# B&R Automation Studio project Mapp6D_Demo
Automation Studio 4.10.3.60 SP; technology packages: mapp6D 1.1.0, mappView 5.12.1

## Configuration Config1

CPU X20CP1685, AutomationRuntime C4.90, Build 4.1.2, Safety 0.0, Vc V4.72.3

### Task classes (Cpu.sw)
```
Cyclic#4:
  Macro <- Macro.prg
  ShuttleGro <- ShuttleGroup.prg
  VirtualShu <- VirtualShuttle1.prg
  Planet <- Planet.prg
Binaries: FWRules, udbdef, TCData, arcoal, arflatprv, arsvcreg, arconfig, User, Role, sysconf, iomap, asfw, ashwac, ashwd, Config_2, Config_1
Libraries: McBase, brsystem, runtime, AsBrStr, McAcp6D, astime, asieccon, fileio
```

### Hardware
```
8YFLM01.0000.00I-1 : 8YFLM01.0000.00I-1 v0.0.0.1  [PLK1 -> X20CP1685.IF3 (NodeNumber=50) [Cable Type=PowerlinkCable, Length=10, Version=1.0.0.3]]
  Supervision = off
X20CP1685 : X20CP1685 v1.4.0.0
  Connector IF2:
    ActivateDevice = 1
    Mode = Manual
    InternetAddress = 192.168.10.7
    SubnetMask = 255.255.255.0
    ActivateSnmp = 2
  Connector IF3:
    CycleTime = 1000
  ConfigurationID = mapp6d_SampleProject_Config1
  UserPartitionSize = 10
  TimerDeviceType = EPLX2X
  TimerDevice = X20CP1685.IF3
  TaskClassIdleTime = 2000
  Cyclic1Duration = 1000
  Cyclic1Tolerance = 0
  Cyclic3Duration = 52000
  Cyclic3Tolerance = 52000
  Cyclic5Duration = 198000
  Cyclic5Tolerance = 198000
  Cyclic7Duration = 1002000
  Cyclic7Tolerance = 1002000
  FileDevice1
  FileDeviceName1 = 6DData
  FileDevicePath1 = C:\6DData
  FtpUser1
  FtpUsername1 = admin
  FtpUserPassword1 = dNmF8ZjP+LmBsEglWtmW9suMlO0FNzgHVeilX4YjqJw=
  FtpUserSalt1 = G7mT75Ku
  FTPAccessRight1 = 0
  FTPdevice1 = ALL
```

### Config_1.assembly6d - X20CP1685/mapp6D/Config_1.assembly6d
```
Element gAssembly6D_1 (Type=assembly6d)
  Simulation6D = SimOn
  Shuttles:
    MaxShuttleCount = 2
    ShuttleIDMode = RealTimeID
    DefaultPosition:
      DefZ = 1.0
      DefRx = 0
      DefRy = 0
      DefRz = 0
    Limits:
      InPlaneLimits:
        InPlaneVelLim = 2
        InPlaneAccLim = 20
        InPlaneEmergDec = 20
      ShortAxLim:
        ShortAxAccLim:
          AccZLim = 10.0
          AccRxLim = 10.0
          AccRyLim = 10.0
          AccRzLim = 10.0
        ShortAxVelLim:
          VelZLim = 0.15
          VelRxLim = 0.1
          VelRyLim = 0.1
          VelRzLim = 0.3
  CyclicChannel6D:
    ReadChannel:
      Xaxis = TRUE
      Yaxis = TRUE
      Zaxis = TRUE
      Rxaxis = TRUE
      Ryaxis = TRUE
      Rzaxis = TRUE
  Fieldbus6D:
    SyncMode6D = ExternalPlkSync
    NodeNumber = 50
  IOMapp:
    Input = ::gComm6D_IN
    Output = ::gComm6D_OUT
  Layout:
    Layout6D[1] = Layout6D_1
```

### Config_2.layout6d - X20CP1685/mapp6D/Config_2.layout6d
```
Element Layout6D_1 (Type=layout6d)
  Segments:
    SegRow = 2
    SegCol = 1
    Segment[1]:
      X = 0
      Y = 0
      Name
      IsMaster = True
    Segment[2]:
      X = 0
      Y = 1
      Name
      IsMaster = False
```

## Configuration Config2

CPU 5APC2100.BY44-000, AutomationRuntime D4.83, Build 4.1.2, Safety 0.0, Vc V4.72.3

### Task classes (Cpu.sw)
```
Cyclic#1 (cycle 1000 us, tolerance 0 us):
  MainCtrl <- MainCtrl.prg
Cyclic#2:
  Macro <- Macro.prg
Cyclic#8 (cycle 5000 us):
  HMI <- HMI.prg
Binaries: FWRules, udbdef, TCData, arcoal, arflatprv, arsvcreg, mvLoader, arconfig, User, Role, sysconf, iomap, asfw, ashwac, ashwd, Config_2, Config_1
Libraries: McBase, brsystem, runtime, AsBrStr, McAcp6D, brdkSTR, MTLookUp, sys_lib, standard, astime, asieccon, fileio, arssl
```

### Hardware
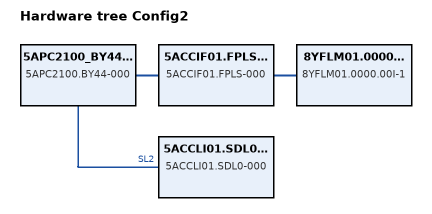
```
5ACCIF01.FPLS-000 : 5ACCIF01.FPLS-000 v2.6.1.0  [SL -> 5APC2100_BY44_000.SL1]
  Connector IF1:
    CycleTime = 1000
5ACCLI01.SDL0-000 : 5ACCLI01.SDL0-000 v2.0.0.0  [SL -> 5APC2100_BY44_000.SL2]
5APC2100_BY44_000 : 5APC2100.BY44-000 v2.1.0.0
  Connector IF3:
    AssignedOperatingSystem = ARemb
    ActivateDevice = 1
    Mode = Manual
    InternetAddress = 192.168.10.7
    SubnetMask = 255.255.255.0
    ActivateSnmp = 2
  Connector IF4:
    AssignedOperatingSystem = ARemb
    ActivateDevice = 1
    Mode = DHCP Server
    InternetAddress = 192.168.0.2
    SubnetMask = 255.255.255.0
    Lease1
    LeaseName1 = 6d_Demo
    LeaseStartAddress1 = 192.168.0.100
    LeaseStopAddress1 = 192.168.0.150
    LeaseSubnetMask1 = 255.255.255.0
  Connector IF5:
    AssignedOperatingSystem = ARemb
  Connector IF6:
    AssignedOperatingSystem = ARemb
  ConfigurationID = mapp6d_SampleProject_Config1
  UserPartitionSize = 10
  UserRamDevice = PCI.1.PPC21xx.SRAM
  UserRamSize = 5000
  RemMemDevice = PCI.1.PPC21xx.SRAM
  RemMemSize = 5000
  RemanentGlobalPvSize = 1000
  TimerDeviceType = EPLX2X
  TimerDevice = 5ACCIF01.FPLS-000.IF1
  TaskClassIdleTime = 2000
  Cyclic1Duration = 1000
  Cyclic1Tolerance = 0
  Cyclic3Duration = 52000
  Cyclic3Tolerance = 52000
  Cyclic5Duration = 198000
  Cyclic5Tolerance = 198000
  Cyclic7Duration = 1002000
  Cyclic7Tolerance = 1002000
  Cyclic8Duration = 5000
  FileDevice1
  FileDeviceName1 = 6DData
  FileDevicePath1 = F:
  FtpUser1
  FtpUsername1 = admin
  FtpUserPassword1 = dNmF8ZjP+LmBsEglWtmW9suMlO0FNzgHVeilX4YjqJw=
  FtpUserSalt1 = G7mT75Ku
  FTPAccessRight1 = 0
  FTPdevice1 = ALL
  ActivateOpcUa = 1
  OpcUaInformationModels_PV_Version = 1
8YFLM01.0000.00I-1 : 8YFLM01.0000.00I-1 v0.0.0.1  [PLK1 -> 5ACCIF01.FPLS-000.IF1 (NodeNumber=50) [Cable Type=PowerlinkCable, Length=10, Version=1.0.0.3]]
  Supervision = off
```

### IoMap.iom - 5APC2100_BY44_000/IoMap.iom
```iecst
VAR_CONFIG
	::gComm6D_IN.Array[0] AT %IW."8YFLM01.0000.00I-1".EPL_FB_IN_0_I2007_S01;
	::gComm6D_IN.Array[1] AT %IW."8YFLM01.0000.00I-1".EPL_FB_IN_1_I2007_S02;
	::gComm6D_IN.Array[2] AT %IW."8YFLM01.0000.00I-1".EPL_FB_IN_2_I2007_S03;
	::gComm6D_IN.Array[3] AT %IW."8YFLM01.0000.00I-1".EPL_FB_IN_3_I2007_S04;
	::gComm6D_IN.Array[4] AT %IW."8YFLM01.0000.00I-1".EPL_FB_IN_4_I2007_S05;
	::gComm6D_IN.Array[5] AT %IW."8YFLM01.0000.00I-1".EPL_FB_IN_5_I2007_S06;
	::gComm6D_IN.Array[6] AT %IW."8YFLM01.0000.00I-1".EPL_FB_IN_6_I2007_S07;
	::gComm6D_IN.Array[7] AT %IW."8YFLM01.0000.00I-1".EPL_FB_IN_7_I2007_S08;
	::gComm6D_IN.Array[8] AT %IW."8YFLM01.0000.00I-1".EPL_FB_IN_8_I2007_S09;
	::gComm6D_IN.Array[9] AT %IW."8YFLM01.0000.00I-1".EPL_FB_IN_9_I2007_S0A;
	::gComm6D_IN.Array[10] AT %IW."8YFLM01.0000.00I-1".EPL_FB_IN_10_I2007_S0B;
	::gComm6D_IN.Array[11] AT %IW."8YFLM01.0000.00I-1".EPL_FB_IN_11_I2007_S0C;
	::gComm6D_IN.Array[12] AT %IW."8YFLM01.0000.00I-1".EPL_FB_IN_12_I2007_S0D;
	::gComm6D_IN.Array[13] AT %IW."8YFLM01.0000.00I-1".EPL_FB_IN_13_I2007_S0E;
	::gComm6D_IN.Array[14] AT %IW."8YFLM01.0000.00I-1".EPL_FB_IN_14_I2007_S0F;
	::gComm6D_IN.Array[15] AT %IW."8YFLM01.0000.00I-1".EPL_FB_IN_15_I2007_S10;
	::gComm6D_IN.Array[16] AT %IW."8YFLM01.0000.00I-1".EPL_FB_IN_16_I2007_S11;
	::gComm6D_IN.Array[17] AT %IW."8YFLM01.0000.00I-1".EPL_FB_IN_17_I2007_S12;
	::gComm6D_IN.Array[18] AT %IW."8YFLM01.0000.00I-1".EPL_FB_IN_18_I2007_S13;
	::gComm6D_IN.Array[19] AT %IW."8YFLM01.0000.00I-1".EPL_FB_IN_19_I2007_S14;
	::gComm6D_IN.Array[20] AT %IW."8YFLM01.0000.00I-1".EPL_FB_IN_20_I2007_S15;
	::gComm6D_IN.Array[21] AT %IW."8YFLM01.0000.00I-1".EPL_FB_IN_21_I2007_S16;
	::gComm6D_IN.Array[22] AT %IW."8YFLM01.0000.00I-1".EPL_FB_IN_22_I2007_S17;
	::gComm6D_IN.Array[23] AT %IW."8YFLM01.0000.00I-1".EPL_FB_IN_23_I2007_S18;
	::gComm6D_IN.Array[24] AT %IW."8YFLM01.0000.00I-1".EPL_FB_IN_24_I2007_S19;
	::gComm6D_IN.Array[25] AT %IW."8YFLM01.0000.00I-1".EPL_FB_IN_25_I2007_S1A;
	::gComm6D_IN.Array[26] AT %IW."8YFLM01.0000.00I-1".EPL_FB_IN_26_I2007_S1B;
	::gComm6D_IN.Array[27] AT %IW."8YFLM01.0000.00I-1".EPL_FB_IN_27_I2007_S1C;
	::gComm6D_IN.Array[28] AT %IW."8YFLM01.0000.00I-1".EPL_FB_IN_28_I2007_S1D;
	::gComm6D_IN.Array[29] AT %IW."8YFLM01.0000.00I-1".EPL_FB_IN_29_I2007_S1E;
	::gComm6D_IN.Array[30] AT %IW."8YFLM01.0000.00I-1".EPL_FB_IN_30_I2007_S1F;
	::gComm6D_IN.Array[31] AT %IW."8YFLM01.0000.00I-1".EPL_FB_IN_31_I2007_S20;
	::gComm6D_IN.Array[32] AT %IW."8YFLM01.0000.00I-1".EPL_FB_IN_32_I2007_S21;
	::gComm6D_IN.Array[33] AT %IW."8YFLM01.0000.00I-1".EPL_FB_IN_33_I2007_S22;
	::gComm6D_IN.Array[34] AT %IW."8YFLM01.0000.00I-1".EPL_FB_IN_34_I2007_S23;
	::gComm6D_IN.Array[35] AT %IW."8YFLM01.0000.00I-1".EPL_FB_IN_35_I2007_S24;
	::gComm6D_IN.Array[36] AT %IW."8YFLM01.0000.00I-1".EPL_FB_IN_36_I2007_S25;
	::gComm6D_IN.Array[37] AT %IW."8YFLM01.0000.00I-1".EPL_FB_IN_37_I2007_S26;
	::gComm6D_IN.Array[38] AT %IW."8YFLM01.0000.00I-1".EPL_FB_IN_38_I2007_S27;
	::gComm6D_IN.Array[39] AT %IW."8YFLM01.0000.00I-1".EPL_FB_IN_39_I2007_S28;
	::gComm6D_IN.Array[40] AT %IW."8YFLM01.0000.00I-1".EPL_FB_IN_40_I2007_S29;
	::gComm6D_IN.Array[41] AT %IW."8YFLM01.0000.00I-1".EPL_FB_IN_41_I2007_S2A;
	::gComm6D_IN.Array[42] AT %IW."8YFLM01.0000.00I-1".EPL_FB_IN_42_I2007_S2B;
	::gComm6D_IN.Array[43] AT %IW."8YFLM01.0000.00I-1".EPL_FB_IN_43_I2007_S2C;
	::gComm6D_IN.Array[44] AT %IW."8YFLM01.0000.00I-1".EPL_FB_IN_44_I2007_S2D;
	::gComm6D_IN.Array[45] AT %IW."8YFLM01.0000.00I-1".EPL_FB_IN_45_I2007_S2E;
	::gComm6D_IN.Array[46] AT %IW."8YFLM01.0000.00I-1".EPL_FB_IN_46_I2007_S2F;
	::gComm6D_IN.Array[47] AT %IW."8YFLM01.0000.00I-1".EPL_FB_IN_47_I2007_S30;
	::gComm6D_IN.Array[48] AT %IW."8YFLM01.0000.00I-1".EPL_FB_IN_48_I2007_S31;
	::gComm6D_IN.Array[49] AT %IW."8YFLM01.0000.00I-1".EPL_FB_IN_49_I2007_S32;
	::gComm6D_IN.Array[50] AT %IW."8YFLM01.0000.00I-1".EPL_FB_IN_50_I2007_S33;
	::gComm6D_IN.Array[51] AT %IW."8YFLM01.0000.00I-1".EPL_FB_IN_51_I2007_S34;
	::gComm6D_IN.Array[52] AT %IW."8YFLM01.0000.00I-1".EPL_FB_IN_52_I2007_S35;
	::gComm6D_IN.Array[53] AT %IW."8YFLM01.0000.00I-1".EPL_FB_IN_53_I2007_S36;
	::gComm6D_IN.Array[54] AT %IW."8YFLM01.0000.00I-1".EPL_FB_IN_54_I2007_S37;
	::gComm6D_IN.Array[55] AT %IW."8YFLM01.0000.00I-1".EPL_FB_IN_55_I2007_S38;
	::gComm6D_IN.Array[56] AT %IW."8YFLM01.0000.00I-1".EPL_FB_IN_56_I2007_S39;
	::gComm6D_IN.Array[57] AT %IW."8YFLM01.0000.00I-1".EPL_FB_IN_57_I2007_S3A;
	::gComm6D_IN.Array[58] AT %IW."8YFLM01.0000.00I-1".EPL_FB_IN_58_I2007_S3B;
	::gComm6D_IN.Array[59] AT %IW."8YFLM01.0000.00I-1".EPL_FB_IN_59_I2007_S3C;
	::gComm6D_IN.Array[60] AT %IW."8YFLM01.0000.00I-1".EPL_FB_IN_60_I2007_S3D;
	::gComm6D_IN.Array[61] AT %IW."8YFLM01.0000.00I-1".EPL_FB_IN_61_I2007_S3E;
	::gComm6D_IN.Array[62] AT %IW."8YFLM01.0000.00I-1".EPL_FB_IN_62_I2007_S3F;
	::gComm6D_IN.Array[63] AT %IW."8YFLM01.0000.00I-1".EPL_FB_IN_63_I2007_S40;
	::gComm6D_IN.Array[64] AT %IW."8YFLM01.0000.00I-1".EPL_FB_IN_64_I2007_S41;
	::gComm6D_IN.Array[65] AT %IW."8YFLM01.0000.00I-1".EPL_FB_IN_65_I2007_S42;
	::gComm6D_IN.Array[66] AT %IW."8YFLM01.0000.00I-1".EPL_FB_IN_66_I2007_S43;
	::gComm6D_IN.Array[67] AT %IW."8YFLM01.0000.00I-1".EPL_FB_IN_67_I2007_S44;
	::gComm6D_IN.Array[68] AT %IW."8YFLM01.0000.00I-1".EPL_FB_IN_68_I2007_S45;
	::gComm6D_IN.Array[69] AT %IW."8YFLM01.0000.00I-1".EPL_FB_IN_69_I2007_S46;
	::gComm6D_IN.Array[70] AT %IW."8YFLM01.0000.00I-1".EPL_FB_IN_70_I2007_S47;
	::gComm6D_IN.Array[71] AT %IW."8YFLM01.0000.00I-1".EPL_FB_IN_71_I2007_S48;
	::gComm6D_IN.Array[72] AT %IW."8YFLM01.0000.00I-1".EPL_FB_IN_72_I2007_S49;
	::gComm6D_IN.Array[73] AT %IW."8YFLM01.0000.00I-1".EPL_FB_IN_73_I2007_S4A;
	::gComm6D_IN.Array[74] AT %IW."8YFLM01.0000.00I-1".EPL_FB_IN_74_I2007_S4B;
	::gComm6D_IN.Array[75] AT %IW."8YFLM01.0000.00I-1".EPL_FB_IN_75_I2007_S4C;
	::gComm6D_IN.Array[76] AT %IW."8YFLM01.0000.00I-1".EPL_FB_IN_76_I2007_S4D;
	::gComm6D_IN.Array[77] AT %IW."8YFLM01.0000.00I-1".EPL_FB_IN_77_I2007_S4E;
	::gComm6D_IN.Array[78] AT %IW."8YFLM01.0000.00I-1".EPL_FB_IN_78_I2007_S4F;
	::gComm6D_IN.Array[79] AT %IW."8YFLM01.0000.00I-1".EPL_FB_IN_79_I2007_S50;
	::gComm6D_IN.Array[80] AT %IW."8YFLM01.0000.00I-1".EPL_FB_IN_80_I2007_S51;
	::gComm6D_IN.Array[81] AT %IW."8YFLM01.0000.00I-1".EPL_FB_IN_81_I2007_S52;
	::gComm6D_IN.Array[82] AT %IW."8YFLM01.0000.00I-1".EPL_FB_IN_82_I2007_S53;
	::gComm6D_IN.Array[83] AT %IW."8YFLM01.0000.00I-1".EPL_FB_IN_83_I2007_S54;
	::gComm6D_IN.Array[84] AT %IW."8YFLM01.0000.00I-1".EPL_FB_IN_84_I2007_S55;
	::gComm6D_IN.Array[85] AT %IW."8YFLM01.0000.00I-1".EPL_FB_IN_85_I2007_S56;
	::gComm6D_IN.Array[86] AT %IW."8YFLM01.0000.00I-1".EPL_FB_IN_86_I2007_S57;
	::gComm6D_IN.Array[87] AT %IW."8YFLM01.0000.00I-1".EPL_FB_IN_87_I2007_S58;
	::gComm6D_IN.Array[88] AT %IW."8YFLM01.0000.00I-1".EPL_FB_IN_88_I2007_S59;
	::gComm6D_IN.Array[89] AT %IW."8YFLM01.0000.00I-1".EPL_FB_IN_89_I2007_S5A;
	::gComm6D_IN.Array[90] AT %IW."8YFLM01.0000.00I-1".EPL_FB_IN_90_I2007_S5B;
	::gComm6D_IN.Array[91] AT %IW."8YFLM01.0000.00I-1".EPL_FB_IN_91_I2007_S5C;
	::gComm6D_IN.Array[92] AT %IW."8YFLM01.0000.00I-1".EPL_FB_IN_92_I2007_S5D;
	::gComm6D_IN.Array[93] AT %IW."8YFLM01.0000.00I-1".EPL_FB_IN_93_I2007_S5E;
	::gComm6D_IN.Array[94] AT %IW."8YFLM01.0000.00I-1".EPL_FB_IN_94_I2007_S5F;
	::gComm6D_IN.Array[95] AT %IW."8YFLM01.0000.00I-1".EPL_FB_IN_95_I2007_S60;
	::gComm6D_IN.Array[96] AT %IW."8YFLM01.0000.00I-1".EPL_FB_IN_96_I2007_S61;
	::gComm6D_IN.Array[97] AT %IW."8YFLM01.0000.00I-1".EPL_FB_IN_97_I2007_S62;
	::gComm6D_IN.Array[98] AT %IW."8YFLM01.0000.00I-1".EPL_FB_IN_98_I2007_S63;
	::gComm6D_IN.Array[99] AT %IW."8YFLM01.0000.00I-1".EPL_FB_IN_99_I2007_S64;
	::gComm6D_IN.Array[100] AT %IW."8YFLM01.0000.00I-1".EPL_FB_IN_100_I2007_S65;
	::gComm6D_IN.Array[101] AT %IW."8YFLM01.0000.00I-1".EPL_FB_IN_101_I2007_S66;
	::gComm6D_IN.Array[102] AT %IW."8YFLM01.0000.00I-1".EPL_FB_IN_102_I2007_S67;
	::gComm6D_IN.Array[103] AT %IW."8YFLM01.0000.00I-1".EPL_FB_IN_103_I2007_S68;
	::gComm6D_IN.Array[104] AT %IW."8YFLM01.0000.00I-1".EPL_FB_IN_104_I2007_S69;
	::gComm6D_IN.Array[105] AT %IW."8YFLM01.0000.00I-1".EPL_FB_IN_105_I2007_S6A;
	::gComm6D_IN.Array[106] AT %IW."8YFLM01.0000.00I-1".EPL_FB_IN_106_I2007_S6B;
	::gComm6D_IN.Array[107] AT %IW."8YFLM01.0000.00I-1".EPL_FB_IN_107_I2007_S6C;
	::gComm6D_IN.Array[108] AT %IW."8YFLM01.0000.00I-1".EPL_FB_IN_108_I2007_S6D;
	::gComm6D_IN.Array[109] AT %IW."8YFLM01.0000.00I-1".EPL_FB_IN_109_I2007_S6E;
	::gComm6D_IN.Array[110] AT %IW."8YFLM01.0000.00I-1".EPL_FB_IN_110_I2007_S6F;
	::gComm6D_IN.Array[111] AT %IW."8YFLM01.0000.00I-1".EPL_FB_IN_111_I2007_S70;
	::gComm6D_IN.Array[112] AT %IW."8YFLM01.0000.00I-1".EPL_FB_IN_112_I2007_S71;
	::gComm6D_IN.Array[113] AT %IW."8YFLM01.0000.00I-1".EPL_FB_IN_113_I2007_S72;
	::gComm6D_IN.Array[114] AT %IW."8YFLM01.0000.00I-1".EPL_FB_IN_114_I2007_S73;
	::gComm6D_IN.Array[115] AT %IW."8YFLM01.0000.00I-1".EPL_FB_IN_115_I2007_S74;
	::gComm6D_IN.Array[116] AT %IW."8YFLM01.0000.00I-1".EPL_FB_IN_116_I2007_S75;
	::gComm6D_IN.Array[117] AT %IW."8YFLM01.0000.00I-1".EPL_FB_IN_117_I2007_S76;
	::gComm6D_IN.Array[118] AT %IW."8YFLM01.0000.00I-1".EPL_FB_IN_118_I2007_S77;
	::gComm6D_IN.Array[119] AT %IW."8YFLM01.0000.00I-1".EPL_FB_IN_119_I2007_S78;
	::gComm6D_IN.Array[120] AT %IW."8YFLM01.0000.00I-1".EPL_FB_IN_120_I2007_S79;
	::gComm6D_IN.Array[121] AT %IW."8YFLM01.0000.00I-1".EPL_FB_IN_121_I2007_S7A;
	::gComm6D_IN.Array[122] AT %IW."8YFLM01.0000.00I-1".EPL_FB_IN_122_I2007_S7B;
	::gComm6D_IN.Array[123] AT %IW."8YFLM01.0000.00I-1".EPL_FB_IN_123_I2007_S7C;
	::gComm6D_IN.Array[124] AT %IW."8YFLM01.0000.00I-1".EPL_FB_IN_124_I2007_S7D;
	::gComm6D_IN.Array[125] AT %IW."8YFLM01.0000.00I-1".EPL_FB_IN_125_I2007_S7E;
	::gComm6D_IN.Array[126] AT %IW."8YFLM01.0000.00I-1".EPL_FB_IN_126_I2007_S7F;
	::gComm6D_IN.Array[127] AT %IW."8YFLM01.0000.00I-1".EPL_FB_IN_127_I2007_S80;
	::gComm6D_IN.Array[128] AT %IW."8YFLM01.0000.00I-1".EPL_FB_IN_128_I2007_S81;
	::gComm6D_IN.Array[129] AT %IW."8YFLM01.0000.00I-1".EPL_FB_IN_129_I2007_S82;
	::gComm6D_IN.Array[130] AT %IW."8YFLM01.0000.00I-1".EPL_FB_IN_130_I2007_S83;
	::gComm6D_IN.Array[131] AT %IW."8YFLM01.0000.00I-1".EPL_FB_IN_131_I2007_S84;
	::gComm6D_IN.Array[132] AT %IW."8YFLM01.0000.00I-1".EPL_FB_IN_132_I2007_S85;
	::gComm6D_IN.Array[133] AT %IW."8YFLM01.0000.00I-1".EPL_FB_IN_133_I2007_S86;
	::gComm6D_IN.Array[134] AT %IW."8YFLM01.0000.00I-1".EPL_FB_IN_134_I2007_S87;
	::gComm6D_IN.Array[135] AT %IW."8YFLM01.0000.00I-1".EPL_FB_IN_135_I2007_S88;
	::gComm6D_IN.Array[136] AT %IW."8YFLM01.0000.00I-1".EPL_FB_IN_136_I2007_S89;
	::gComm6D_IN.Array[137] AT %IW."8YFLM01.0000.00I-1".EPL_FB_IN_137_I2007_S8A;
	::gComm6D_IN.Array[138] AT %IW."8YFLM01.0000.00I-1".EPL_FB_IN_138_I2007_S8B;
	::gComm6D_IN.Array[139] AT %IW."8YFLM01.0000.00I-1".EPL_FB_IN_139_I2007_S8C;
	::gComm6D_IN.Array[140] AT %IW."8YFLM01.0000.00I-1".EPL_FB_IN_140_I2007_S8D;
	::gComm6D_IN.Array[141] AT %IW."8YFLM01.0000.00I-1".EPL_FB_IN_141_I2007_S8E;
	::gComm6D_IN.Array[142] AT %IW."8YFLM01.0000.00I-1".EPL_FB_IN_142_I2007_S8F;
	::gComm6D_IN.Array[143] AT %IW."8YFLM01.0000.00I-1".EPL_FB_IN_143_I2007_S90;
	::gComm6D_IN.Array[144] AT %IW."8YFLM01.0000.00I-1".EPL_FB_IN_144_I2007_S91;
	::gComm6D_IN.Array[145] AT %IW."8YFLM01.0000.00I-1".EPL_FB_IN_145_I2007_S92;
	::gComm6D_IN.Array[146] AT %IW."8YFLM01.0000.00I-1".EPL_FB_IN_146_I2007_S93;
	::gComm6D_IN.Array[147] AT %IW."8YFLM01.0000.00I-1".EPL_FB_IN_147_I2007_S94;
	::gComm6D_IN.Array[148] AT %IW."8YFLM01.0000.00I-1".EPL_FB_IN_148_I2007_S95;
	::gComm6D_IN.Array[149] AT %IW."8YFLM01.0000.00I-1".EPL_FB_IN_149_I2007_S96;
	::gComm6D_IN.Array[150] AT %IW."8YFLM01.0000.00I-1".EPL_FB_IN_150_I2007_S97;
	::gComm6D_IN.Array[151] AT %IW."8YFLM01.0000.00I-1".EPL_FB_IN_151_I2007_S98;
	::gComm6D_IN.Array[152] AT %IW."8YFLM01.0000.00I-1".EPL_FB_IN_152_I2007_S99;
	::gComm6D_IN.Array[153] AT %IW."8YFLM01.0000.00I-1".EPL_FB_IN_153_I2007_S9A;
	::gComm6D_IN.Array[154] AT %IW."8YFLM01.0000.00I-1".EPL_FB_IN_154_I2007_S9B;
	::gComm6D_IN.Array[155] AT %IW."8YFLM01.0000.00I-1".EPL_FB_IN_155_I2007_S9C;
	::gComm6D_IN.Array[156] AT %IW."8YFLM01.0000.00I-1".EPL_FB_IN_156_I2007_S9D;
	::gComm6D_IN.Array[157] AT %IW."8YFLM01.0000.00I-1".EPL_FB_IN_157_I2007_S9E;
	::gComm6D_IN.Array[158] AT %IW."8YFLM01.0000.00I-1".EPL_FB_IN_158_I2007_S9F;
	::gComm6D_IN.Array[159] AT %IW."8YFLM01.0000.00I-1".EPL_FB_IN_159_I2007_SA0;
	::gComm6D_IN.Array[160] AT %IW."8YFLM01.0000.00I-1".EPL_FB_IN_160_I2007_SA1;
	::gComm6D_IN.Array[161] AT %IW."8YFLM01.0000.00I-1".EPL_FB_IN_161_I2007_SA2;
	::gComm6D_IN.Array[162] AT %IW."8YFLM01.0000.00I-1".EPL_FB_IN_162_I2007_SA3;
	::gComm6D_IN.Array[163] AT %IW."8YFLM01.0000.00I-1".EPL_FB_IN_163_I2007_SA4;
	::gComm6D_IN.Array[164] AT %IW."8YFLM01.0000.00I-1".EPL_FB_IN_164_I2007_SA5;
	::gComm6D_IN.Array[165] AT %IW."8YFLM01.0000.00I-1".EPL_FB_IN_165_I2007_SA6;
	::gComm6D_IN.Array[166] AT %IW."8YFLM01.0000.00I-1".EPL_FB_IN_166_I2007_SA7;
	::gComm6D_IN.Array[167] AT %IW."8YFLM01.0000.00I-1".EPL_FB_IN_167_I2007_SA8;
	::gComm6D_IN.Array[168] AT %IW."8YFLM01.0000.00I-1".EPL_FB_IN_168_I2007_SA9;
	::gComm6D_IN.Array[169] AT %IW."8YFLM01.0000.00I-1".EPL_FB_IN_169_I2007_SAA;
	::gComm6D_IN.Array[170] AT %IW."8YFLM01.0000.00I-1".EPL_FB_IN_170_I2007_SAB;
	::gComm6D_IN.Array[171] AT %IW."8YFLM01.0000.00I-1".EPL_FB_IN_171_I2007_SAC;
	::gComm6D_IN.Array[172] AT %IW."8YFLM01.0000.00I-1".EPL_FB_IN_172_I2007_SAD;
	::gComm6D_IN.Array[173] AT %IW."8YFLM01.0000.00I-1".EPL_FB_IN_173_I2007_SAE;
	::gComm6D_IN.Array[174] AT %IW."8YFLM01.0000.00I-1".EPL_FB_IN_174_I2007_SAF;
	::gComm6D_IN.Array[175] AT %IW."8YFLM01.0000.00I-1".EPL_FB_IN_175_I2007_SB0;
	::gComm6D_IN.Array[176] AT %IW."8YFLM01.0000.00I-1".EPL_FB_IN_176_I2007_SB1;
	::gComm6D_IN.Array[177] AT %IW."8YFLM01.0000.00I-1".EPL_FB_IN_177_I2007_SB2;
	::gComm6D_IN.Array[178] AT %IW."8YFLM01.0000.00I-1".EPL_FB_IN_178_I2007_SB3;
	::gComm6D_IN.Array[179] AT %IW."8YFLM01.0000.00I-1".EPL_FB_IN_179_I2007_SB4;
	::gComm6D_IN.Array[180] AT %IW."8YFLM01.0000.00I-1".EPL_FB_IN_180_I2007_SB5;
	::gComm6D_IN.Array[181] AT %IW."8YFLM01.0000.00I-1".EPL_FB_IN_181_I2007_SB6;
	::gComm6D_IN.Array[182] AT %IW."8YFLM01.0000.00I-1".EPL_FB_IN_182_I2007_SB7;
	::gComm6D_IN.Array[183] AT %IW."8YFLM01.0000.00I-1".EPL_FB_IN_183_I2007_SB8;
	::gComm6D_IN.Array[184] AT %IW."8YFLM01.0000.00I-1".EPL_FB_IN_184_I2007_SB9;
	::gComm6D_IN.Array[185] AT %IW."8YFLM01.0000.00I-1".EPL_FB_IN_185_I2007_SBA;
	::gComm6D_IN.Array[186] AT %IW."8YFLM01.0000.00I-1".EPL_FB_IN_186_I2007_SBB;
	::gComm6D_IN.Array[187] AT %IW."8YFLM01.0000.00I-1".EPL_FB_IN_187_I2007_SBC;
	::gComm6D_IN.Array[188] AT %IW."8YFLM01.0000.00I-1".EPL_FB_IN_188_I2007_SBD;
	::gComm6D_IN.Array[189] AT %IW."8YFLM01.0000.00I-1".EPL_FB_IN_189_I2007_SBE;
	::gComm6D_IN.Array[190] AT %IW."8YFLM01.0000.00I-1".EPL_FB_IN_190_I2007_SBF;
	::gComm6D_IN.Array[191] AT %IW."8YFLM01.0000.00I-1".EPL_FB_IN_191_I2007_SC0;
	::gComm6D_IN.Array[192] AT %IW."8YFLM01.0000.00I-1".EPL_FB_IN_192_I2007_SC1;
	::gComm6D_IN.Array[193] AT %IW."8YFLM01.0000.00I-1".EPL_FB_IN_193_I2007_SC2;
	::gComm6D_IN.Array[194] AT %IW."8YFLM01.0000.00I-1".EPL_FB_IN_194_I2007_SC3;
	::gComm6D_IN.Array[195] AT %IW."8YFLM01.0000.00I-1".EPL_FB_IN_195_I2007_SC4;
	::gComm6D_IN.Array[196] AT %IW."8YFLM01.0000.00I-1".EPL_FB_IN_196_I2007_SC5;
	::gComm6D_IN.Array[197] AT %IW."8YFLM01.0000.00I-1".EPL_FB_IN_197_I2007_SC6;
	::gComm6D_IN.Array[198] AT %IW."8YFLM01.0000.00I-1".EPL_FB_IN_198_I2007_SC7;
	::gComm6D_IN.Array[199] AT %IW."8YFLM01.0000.00I-1".EPL_FB_IN_199_I2007_SC8;
	::gComm6D_OUT.Array[0] AT %QW."8YFLM01.0000.00I-1".EPL_FB_OUT_0_I2008_S01Out;
	::gComm6D_OUT.Array[1] AT %QW."8YFLM01.0000.00I-1".EPL_FB_OUT_1_I2008_S02Out;
	::gComm6D_OUT.Array[2] AT %QW."8YFLM01.0000.00I-1".EPL_FB_OUT_2_I2008_S03Out;
	::gComm6D_OUT.Array[3] AT %QW."8YFLM01.0000.00I-1".EPL_FB_OUT_3_I2008_S04Out;
	::gComm6D_OUT.Array[4] AT %QW."8YFLM01.0000.00I-1".EPL_FB_OUT_4_I2008_S05Out;
	::gComm6D_OUT.Array[5] AT %QW."8YFLM01.0000.00I-1".EPL_FB_OUT_5_I2008_S06Out;
	::gComm6D_OUT.Array[6] AT %QW."8YFLM01.0000.00I-1".EPL_FB_OUT_6_I2008_S07Out;
	::gComm6D_OUT.Array[7] AT %QW."8YFLM01.0000.00I-1".EPL_FB_OUT_7_I2008_S08Out;
	::gComm6D_OUT.Array[8] AT %QW."8YFLM01.0000.00I-1".EPL_FB_OUT_8_I2008_S09Out;
	::gComm6D_OUT.Array[9] AT %QW."8YFLM01.0000.00I-1".EPL_FB_OUT_9_I2008_S0AOut;
	::gComm6D_OUT.Array[10] AT %QW."8YFLM01.0000.00I-1".EPL_FB_OUT_10_I2008_S0BOut;
	::gComm6D_OUT.Array[11] AT %QW."8YFLM01.0000.00I-1".EPL_FB_OUT_11_I2008_S0COut;
	::gComm6D_OUT.Array[12] AT %QW."8YFLM01.0000.00I-1".EPL_FB_OUT_12_I2008_S0DOut;
	::gComm6D_OUT.Array[13] AT %QW."8YFLM01.0000.00I-1".EPL_FB_OUT_13_I2008_S0EOut;
	::gComm6D_OUT.Array[14] AT %QW."8YFLM01.0000.00I-1".EPL_FB_OUT_14_I2008_S0FOut;
	::gComm6D_OUT.Array[15] AT %QW."8YFLM01.0000.00I-1".EPL_FB_OUT_15_I2008_S10Out;
	::gComm6D_OUT.Array[16] AT %QW."8YFLM01.0000.00I-1".EPL_FB_OUT_16_I2008_S11Out;
	::gComm6D_OUT.Array[17] AT %QW."8YFLM01.0000.00I-1".EPL_FB_OUT_17_I2008_S12Out;
	::gComm6D_OUT.Array[18] AT %QW."8YFLM01.0000.00I-1".EPL_FB_OUT_18_I2008_S13Out;
	::gComm6D_OUT.Array[19] AT %QW."8YFLM01.0000.00I-1".EPL_FB_OUT_19_I2008_S14Out;
	::gComm6D_OUT.Array[20] AT %QW."8YFLM01.0000.00I-1".EPL_FB_OUT_20_I2008_S15Out;
	::gComm6D_OUT.Array[21] AT %QW."8YFLM01.0000.00I-1".EPL_FB_OUT_21_I2008_S16Out;
	::gComm6D_OUT.Array[22] AT %QW."8YFLM01.0000.00I-1".EPL_FB_OUT_22_I2008_S17Out;
	::gComm6D_OUT.Array[23] AT %QW."8YFLM01.0000.00I-1".EPL_FB_OUT_23_I2008_S18Out;
	::gComm6D_OUT.Array[24] AT %QW."8YFLM01.0000.00I-1".EPL_FB_OUT_24_I2008_S19Out;
	::gComm6D_OUT.Array[25] AT %QW."8YFLM01.0000.00I-1".EPL_FB_OUT_25_I2008_S1AOut;
	::gComm6D_OUT.Array[26] AT %QW."8YFLM01.0000.00I-1".EPL_FB_OUT_26_I2008_S1BOut;
	::gComm6D_OUT.Array[27] AT %QW."8YFLM01.0000.00I-1".EPL_FB_OUT_27_I2008_S1COut;
	::gComm6D_OUT.Array[28] AT %QW."8YFLM01.0000.00I-1".EPL_FB_OUT_28_I2008_S1DOut;
	::gComm6D_OUT.Array[29] AT %QW."8YFLM01.0000.00I-1".EPL_FB_OUT_29_I2008_S1EOut;
	::gComm6D_OUT.Array[30] AT %QW."8YFLM01.0000.00I-1".EPL_FB_OUT_30_I2008_S1FOut;
	::gComm6D_OUT.Array[31] AT %QW."8YFLM01.0000.00I-1".EPL_FB_OUT_31_I2008_S20Out;
	::gComm6D_OUT.Array[32] AT %QW."8YFLM01.0000.00I-1".EPL_FB_OUT_32_I2008_S21Out;
	::gComm6D_OUT.Array[33] AT %QW."8YFLM01.0000.00I-1".EPL_FB_OUT_33_I2008_S22Out;
	::gComm6D_OUT.Array[34] AT %QW."8YFLM01.0000.00I-1".EPL_FB_OUT_34_I2008_S23Out;
	::gComm6D_OUT.Array[35] AT %QW."8YFLM01.0000.00I-1".EPL_FB_OUT_35_I2008_S24Out;
	::gComm6D_OUT.Array[36] AT %QW."8YFLM01.0000.00I-1".EPL_FB_OUT_36_I2008_S25Out;
	::gComm6D_OUT.Array[37] AT %QW."8YFLM01.0000.00I-1".EPL_FB_OUT_37_I2008_S26Out;
	::gComm6D_OUT.Array[38] AT %QW."8YFLM01.0000.00I-1".EPL_FB_OUT_38_I2008_S27Out;
	::gComm6D_OUT.Array[39] AT %QW."8YFLM01.0000.00I-1".EPL_FB_OUT_39_I2008_S28Out;
	::gComm6D_OUT.Array[40] AT %QW."8YFLM01.0000.00I-1".EPL_FB_OUT_40_I2008_S29Out;
	::gComm6D_OUT.Array[41] AT %QW."8YFLM01.0000.00I-1".EPL_FB_OUT_41_I2008_S2AOut;
	::gComm6D_OUT.Array[42] AT %QW."8YFLM01.0000.00I-1".EPL_FB_OUT_42_I2008_S2BOut;
	::gComm6D_OUT.Array[43] AT %QW."8YFLM01.0000.00I-1".EPL_FB_OUT_43_I2008_S2COut;
	::gComm6D_OUT.Array[44] AT %QW."8YFLM01.0000.00I-1".EPL_FB_OUT_44_I2008_S2DOut;
	::gComm6D_OUT.Array[45] AT %QW."8YFLM01.0000.00I-1".EPL_FB_OUT_45_I2008_S2EOut;
	::gComm6D_OUT.Array[46] AT %QW."8YFLM01.0000.00I-1".EPL_FB_OUT_46_I2008_S2FOut;
	::gComm6D_OUT.Array[47] AT %QW."8YFLM01.0000.00I-1".EPL_FB_OUT_47_I2008_S30Out;
	::gComm6D_OUT.Array[48] AT %QW."8YFLM01.0000.00I-1".EPL_FB_OUT_48_I2008_S31Out;
	::gComm6D_OUT.Array[49] AT %QW."8YFLM01.0000.00I-1".EPL_FB_OUT_49_I2008_S32Out;
	::gComm6D_OUT.Array[50] AT %QW."8YFLM01.0000.00I-1".EPL_FB_OUT_50_I2008_S33Out;
	::gComm6D_OUT.Array[51] AT %QW."8YFLM01.0000.00I-1".EPL_FB_OUT_51_I2008_S34Out;
	::gComm6D_OUT.Array[52] AT %QW."8YFLM01.0000.00I-1".EPL_FB_OUT_52_I2008_S35Out;
	::gComm6D_OUT.Array[53] AT %QW."8YFLM01.0000.00I-1".EPL_FB_OUT_53_I2008_S36Out;
	::gComm6D_OUT.Array[54] AT %QW."8YFLM01.0000.00I-1".EPL_FB_OUT_54_I2008_S37Out;
	::gComm6D_OUT.Array[55] AT %QW."8YFLM01.0000.00I-1".EPL_FB_OUT_55_I2008_S38Out;
	::gComm6D_OUT.Array[56] AT %QW."8YFLM01.0000.00I-1".EPL_FB_OUT_56_I2008_S39Out;
	::gComm6D_OUT.Array[57] AT %QW."8YFLM01.0000.00I-1".EPL_FB_OUT_57_I2008_S3AOut;
	::gComm6D_OUT.Array[58] AT %QW."8YFLM01.0000.00I-1".EPL_FB_OUT_58_I2008_S3BOut;
	::gComm6D_OUT.Array[59] AT %QW."8YFLM01.0000.00I-1".EPL_FB_OUT_59_I2008_S3COut;
	::gComm6D_OUT.Array[60] AT %QW."8YFLM01.0000.00I-1".EPL_FB_OUT_60_I2008_S3DOut;
	::gComm6D_OUT.Array[61] AT %QW."8YFLM01.0000.00I-1".EPL_FB_OUT_61_I2008_S3EOut;
	::gComm6D_OUT.Array[62] AT %QW."8YFLM01.0000.00I-1".EPL_FB_OUT_62_I2008_S3FOut;
	::gComm6D_OUT.Array[63] AT %QW."8YFLM01.0000.00I-1".EPL_FB_OUT_63_I2008_S40Out;
	::gComm6D_OUT.Array[64] AT %QW."8YFLM01.0000.00I-1".EPL_FB_OUT_64_I2008_S41Out;
	::gComm6D_OUT.Array[65] AT %QW."8YFLM01.0000.00I-1".EPL_FB_OUT_65_I2008_S42Out;
	::gComm6D_OUT.Array[66] AT %QW."8YFLM01.0000.00I-1".EPL_FB_OUT_66_I2008_S43Out;
	::gComm6D_OUT.Array[67] AT %QW."8YFLM01.0000.00I-1".EPL_FB_OUT_67_I2008_S44Out;
	::gComm6D_OUT.Array[68] AT %QW."8YFLM01.0000.00I-1".EPL_FB_OUT_68_I2008_S45Out;
	::gComm6D_OUT.Array[69] AT %QW."8YFLM01.0000.00I-1".EPL_FB_OUT_69_I2008_S46Out;
	::gComm6D_OUT.Array[70] AT %QW."8YFLM01.0000.00I-1".EPL_FB_OUT_70_I2008_S47Out;
	::gComm6D_OUT.Array[71] AT %QW."8YFLM01.0000.00I-1".EPL_FB_OUT_71_I2008_S48Out;
	::gComm6D_OUT.Array[72] AT %QW."8YFLM01.0000.00I-1".EPL_FB_OUT_72_I2008_S49Out;
	::gComm6D_OUT.Array[73] AT %QW."8YFLM01.0000.00I-1".EPL_FB_OUT_73_I2008_S4AOut;
	::gComm6D_OUT.Array[74] AT %QW."8YFLM01.0000.00I-1".EPL_FB_OUT_74_I2008_S4BOut;
	::gComm6D_OUT.Array[75] AT %QW."8YFLM01.0000.00I-1".EPL_FB_OUT_75_I2008_S4COut;
	::gComm6D_OUT.Array[76] AT %QW."8YFLM01.0000.00I-1".EPL_FB_OUT_76_I2008_S4DOut;
	::gComm6D_OUT.Array[77] AT %QW."8YFLM01.0000.00I-1".EPL_FB_OUT_77_I2008_S4EOut;
	::gComm6D_OUT.Array[78] AT %QW."8YFLM01.0000.00I-1".EPL_FB_OUT_78_I2008_S4FOut;
	::gComm6D_OUT.Array[79] AT %QW."8YFLM01.0000.00I-1".EPL_FB_OUT_79_I2008_S50Out;
	::gComm6D_OUT.Array[80] AT %QW."8YFLM01.0000.00I-1".EPL_FB_OUT_80_I2008_S51Out;
	::gComm6D_OUT.Array[81] AT %QW."8YFLM01.0000.00I-1".EPL_FB_OUT_81_I2008_S52Out;
	::gComm6D_OUT.Array[82] AT %QW."8YFLM01.0000.00I-1".EPL_FB_OUT_82_I2008_S53Out;
	::gComm6D_OUT.Array[83] AT %QW."8YFLM01.0000.00I-1".EPL_FB_OUT_83_I2008_S54Out;
	::gComm6D_OUT.Array[84] AT %QW."8YFLM01.0000.00I-1".EPL_FB_OUT_84_I2008_S55Out;
	::gComm6D_OUT.Array[85] AT %QW."8YFLM01.0000.00I-1".EPL_FB_OUT_85_I2008_S56Out;
	::gComm6D_OUT.Array[86] AT %QW."8YFLM01.0000.00I-1".EPL_FB_OUT_86_I2008_S57Out;
	::gComm6D_OUT.Array[87] AT %QW."8YFLM01.0000.00I-1".EPL_FB_OUT_87_I2008_S58Out;
	::gComm6D_OUT.Array[88] AT %QW."8YFLM01.0000.00I-1".EPL_FB_OUT_88_I2008_S59Out;
	::gComm6D_OUT.Array[89] AT %QW."8YFLM01.0000.00I-1".EPL_FB_OUT_89_I2008_S5AOut;
	::gComm6D_OUT.Array[90] AT %QW."8YFLM01.0000.00I-1".EPL_FB_OUT_90_I2008_S5BOut;
	::gComm6D_OUT.Array[91] AT %QW."8YFLM01.0000.00I-1".EPL_FB_OUT_91_I2008_S5COut;
	::gComm6D_OUT.Array[92] AT %QW."8YFLM01.0000.00I-1".EPL_FB_OUT_92_I2008_S5DOut;
	::gComm6D_OUT.Array[93] AT %QW."8YFLM01.0000.00I-1".EPL_FB_OUT_93_I2008_S5EOut;
	::gComm6D_OUT.Array[94] AT %QW."8YFLM01.0000.00I-1".EPL_FB_OUT_94_I2008_S5FOut;
	::gComm6D_OUT.Array[95] AT %QW."8YFLM01.0000.00I-1".EPL_FB_OUT_95_I2008_S60Out;
	::gComm6D_OUT.Array[96] AT %QW."8YFLM01.0000.00I-1".EPL_FB_OUT_96_I2008_S61Out;
	::gComm6D_OUT.Array[97] AT %QW."8YFLM01.0000.00I-1".EPL_FB_OUT_97_I2008_S62Out;
	::gComm6D_OUT.Array[98] AT %QW."8YFLM01.0000.00I-1".EPL_FB_OUT_98_I2008_S63Out;
	::gComm6D_OUT.Array[99] AT %QW."8YFLM01.0000.00I-1".EPL_FB_OUT_99_I2008_S64Out;
	::gComm6D_OUT.Array[100] AT %QW."8YFLM01.0000.00I-1".EPL_FB_OUT_100_I2008_S65Out;
	::gComm6D_OUT.Array[101] AT %QW."8YFLM01.0000.00I-1".EPL_FB_OUT_101_I2008_S66Out;
	::gComm6D_OUT.Array[102] AT %QW."8YFLM01.0000.00I-1".EPL_FB_OUT_102_I2008_S67Out;
	::gComm6D_OUT.Array[103] AT %QW."8YFLM01.0000.00I-1".EPL_FB_OUT_103_I2008_S68Out;
	::gComm6D_OUT.Array[104] AT %QW."8YFLM01.0000.00I-1".EPL_FB_OUT_104_I2008_S69Out;
	::gComm6D_OUT.Array[105] AT %QW."8YFLM01.0000.00I-1".EPL_FB_OUT_105_I2008_S6AOut;
	::gComm6D_OUT.Array[106] AT %QW."8YFLM01.0000.00I-1".EPL_FB_OUT_106_I2008_S6BOut;
	::gComm6D_OUT.Array[107] AT %QW."8YFLM01.0000.00I-1".EPL_FB_OUT_107_I2008_S6COut;
	::gComm6D_OUT.Array[108] AT %QW."8YFLM01.0000.00I-1".EPL_FB_OUT_108_I2008_S6DOut;
	::gComm6D_OUT.Array[109] AT %QW."8YFLM01.0000.00I-1".EPL_FB_OUT_109_I2008_S6EOut;
	::gComm6D_OUT.Array[110] AT %QW."8YFLM01.0000.00I-1".EPL_FB_OUT_110_I2008_S6FOut;
	::gComm6D_OUT.Array[111] AT %QW."8YFLM01.0000.00I-1".EPL_FB_OUT_111_I2008_S70Out;
	::gComm6D_OUT.Array[112] AT %QW."8YFLM01.0000.00I-1".EPL_FB_OUT_112_I2008_S71Out;
	::gComm6D_OUT.Array[113] AT %QW."8YFLM01.0000.00I-1".EPL_FB_OUT_113_I2008_S72Out;
	::gComm6D_OUT.Array[114] AT %QW."8YFLM01.0000.00I-1".EPL_FB_OUT_114_I2008_S73Out;
	::gComm6D_OUT.Array[115] AT %QW."8YFLM01.0000.00I-1".EPL_FB_OUT_115_I2008_S74Out;
	::gComm6D_OUT.Array[116] AT %QW."8YFLM01.0000.00I-1".EPL_FB_OUT_116_I2008_S75Out;
	::gComm6D_OUT.Array[117] AT %QW."8YFLM01.0000.00I-1".EPL_FB_OUT_117_I2008_S76Out;
	::gComm6D_OUT.Array[118] AT %QW."8YFLM01.0000.00I-1".EPL_FB_OUT_118_I2008_S77Out;
	::gComm6D_OUT.Array[119] AT %QW."8YFLM01.0000.00I-1".EPL_FB_OUT_119_I2008_S78Out;
	::gComm6D_OUT.Array[120] AT %QW."8YFLM01.0000.00I-1".EPL_FB_OUT_120_I2008_S79Out;
	::gComm6D_OUT.Array[121] AT %QW."8YFLM01.0000.00I-1".EPL_FB_OUT_121_I2008_S7AOut;
	::gComm6D_OUT.Array[122] AT %QW."8YFLM01.0000.00I-1".EPL_FB_OUT_122_I2008_S7BOut;
	::gComm6D_OUT.Array[123] AT %QW."8YFLM01.0000.00I-1".EPL_FB_OUT_123_I2008_S7COut;
	::gComm6D_OUT.Array[124] AT %QW."8YFLM01.0000.00I-1".EPL_FB_OUT_124_I2008_S7DOut;
	::gComm6D_OUT.Array[125] AT %QW."8YFLM01.0000.00I-1".EPL_FB_OUT_125_I2008_S7EOut;
	::gComm6D_OUT.Array[126] AT %QW."8YFLM01.0000.00I-1".EPL_FB_OUT_126_I2008_S7FOut;
	::gComm6D_OUT.Array[127] AT %QW."8YFLM01.0000.00I-1".EPL_FB_OUT_127_I2008_S80Out;
	::gComm6D_OUT.Array[128] AT %QW."8YFLM01.0000.00I-1".EPL_FB_OUT_128_I2008_S81Out;
	::gComm6D_OUT.Array[129] AT %QW."8YFLM01.0000.00I-1".EPL_FB_OUT_129_I2008_S82Out;
	::gComm6D_OUT.Array[130] AT %QW."8YFLM01.0000.00I-1".EPL_FB_OUT_130_I2008_S83Out;
	::gComm6D_OUT.Array[131] AT %QW."8YFLM01.0000.00I-1".EPL_FB_OUT_131_I2008_S84Out;
	::gComm6D_OUT.Array[132] AT %QW."8YFLM01.0000.00I-1".EPL_FB_OUT_132_I2008_S85Out;
	::gComm6D_OUT.Array[133] AT %QW."8YFLM01.0000.00I-1".EPL_FB_OUT_133_I2008_S86Out;
	::gComm6D_OUT.Array[134] AT %QW."8YFLM01.0000.00I-1".EPL_FB_OUT_134_I2008_S87Out;
	::gComm6D_OUT.Array[135] AT %QW."8YFLM01.0000.00I-1".EPL_FB_OUT_135_I2008_S88Out;
	::gComm6D_OUT.Array[136] AT %QW."8YFLM01.0000.00I-1".EPL_FB_OUT_136_I2008_S89Out;
	::gComm6D_OUT.Array[137] AT %QW."8YFLM01.0000.00I-1".EPL_FB_OUT_137_I2008_S8AOut;
	::gComm6D_OUT.Array[138] AT %QW."8YFLM01.0000.00I-1".EPL_FB_OUT_138_I2008_S8BOut;
	::gComm6D_OUT.Array[139] AT %QW."8YFLM01.0000.00I-1".EPL_FB_OUT_139_I2008_S8COut;
	::gComm6D_OUT.Array[140] AT %QW."8YFLM01.0000.00I-1".EPL_FB_OUT_140_I2008_S8DOut;
	::gComm6D_OUT.Array[141] AT %QW."8YFLM01.0000.00I-1".EPL_FB_OUT_141_I2008_S8EOut;
	::gComm6D_OUT.Array[142] AT %QW."8YFLM01.0000.00I-1".EPL_FB_OUT_142_I2008_S8FOut;
	::gComm6D_OUT.Array[143] AT %QW."8YFLM01.0000.00I-1".EPL_FB_OUT_143_I2008_S90Out;
	::gComm6D_OUT.Array[144] AT %QW."8YFLM01.0000.00I-1".EPL_FB_OUT_144_I2008_S91Out;
	::gComm6D_OUT.Array[145] AT %QW."8YFLM01.0000.00I-1".EPL_FB_OUT_145_I2008_S92Out;
	::gComm6D_OUT.Array[146] AT %QW."8YFLM01.0000.00I-1".EPL_FB_OUT_146_I2008_S93Out;
	::gComm6D_OUT.Array[147] AT %QW."8YFLM01.0000.00I-1".EPL_FB_OUT_147_I2008_S94Out;
	::gComm6D_OUT.Array[148] AT %QW."8YFLM01.0000.00I-1".EPL_FB_OUT_148_I2008_S95Out;
	::gComm6D_OUT.Array[149] AT %QW."8YFLM01.0000.00I-1".EPL_FB_OUT_149_I2008_S96Out;
	::gComm6D_OUT.Array[150] AT %QW."8YFLM01.0000.00I-1".EPL_FB_OUT_150_I2008_S97Out;
	::gComm6D_OUT.Array[151] AT %QW."8YFLM01.0000.00I-1".EPL_FB_OUT_151_I2008_S98Out;
	::gComm6D_OUT.Array[152] AT %QW."8YFLM01.0000.00I-1".EPL_FB_OUT_152_I2008_S99Out;
	::gComm6D_OUT.Array[153] AT %QW."8YFLM01.0000.00I-1".EPL_FB_OUT_153_I2008_S9AOut;
	::gComm6D_OUT.Array[154] AT %QW."8YFLM01.0000.00I-1".EPL_FB_OUT_154_I2008_S9BOut;
	::gComm6D_OUT.Array[155] AT %QW."8YFLM01.0000.00I-1".EPL_FB_OUT_155_I2008_S9COut;
	::gComm6D_OUT.Array[156] AT %QW."8YFLM01.0000.00I-1".EPL_FB_OUT_156_I2008_S9DOut;
	::gComm6D_OUT.Array[157] AT %QW."8YFLM01.0000.00I-1".EPL_FB_OUT_157_I2008_S9EOut;
	::gComm6D_OUT.Array[158] AT %QW."8YFLM01.0000.00I-1".EPL_FB_OUT_158_I2008_S9FOut;
	::gComm6D_OUT.Array[159] AT %QW."8YFLM01.0000.00I-1".EPL_FB_OUT_159_I2008_SA0Out;
	::gComm6D_OUT.Array[160] AT %QW."8YFLM01.0000.00I-1".EPL_FB_OUT_160_I2008_SA1Out;
	::gComm6D_OUT.Array[161] AT %QW."8YFLM01.0000.00I-1".EPL_FB_OUT_161_I2008_SA2Out;
	::gComm6D_OUT.Array[162] AT %QW."8YFLM01.0000.00I-1".EPL_FB_OUT_162_I2008_SA3Out;
	::gComm6D_OUT.Array[163] AT %QW."8YFLM01.0000.00I-1".EPL_FB_OUT_163_I2008_SA4Out;
	::gComm6D_OUT.Array[164] AT %QW."8YFLM01.0000.00I-1".EPL_FB_OUT_164_I2008_SA5Out;
	::gComm6D_OUT.Array[165] AT %QW."8YFLM01.0000.00I-1".EPL_FB_OUT_165_I2008_SA6Out;
	::gComm6D_OUT.Array[166] AT %QW."8YFLM01.0000.00I-1".EPL_FB_OUT_166_I2008_SA7Out;
	::gComm6D_OUT.Array[167] AT %QW."8YFLM01.0000.00I-1".EPL_FB_OUT_167_I2008_SA8Out;
	::gComm6D_OUT.Array[168] AT %QW."8YFLM01.0000.00I-1".EPL_FB_OUT_168_I2008_SA9Out;
	::gComm6D_OUT.Array[169] AT %QW."8YFLM01.0000.00I-1".EPL_FB_OUT_169_I2008_SAAOut;
	::gComm6D_OUT.Array[170] AT %QW."8YFLM01.0000.00I-1".EPL_FB_OUT_170_I2008_SABOut;
	::gComm6D_OUT.Array[171] AT %QW."8YFLM01.0000.00I-1".EPL_FB_OUT_171_I2008_SACOut;
	::gComm6D_OUT.Array[172] AT %QW."8YFLM01.0000.00I-1".EPL_FB_OUT_172_I2008_SADOut;
	::gComm6D_OUT.Array[173] AT %QW."8YFLM01.0000.00I-1".EPL_FB_OUT_173_I2008_SAEOut;
	::gComm6D_OUT.Array[174] AT %QW."8YFLM01.0000.00I-1".EPL_FB_OUT_174_I2008_SAFOut;
	::gComm6D_OUT.Array[175] AT %QW."8YFLM01.0000.00I-1".EPL_FB_OUT_175_I2008_SB0Out;
	::gComm6D_OUT.Array[176] AT %QW."8YFLM01.0000.00I-1".EPL_FB_OUT_176_I2008_SB1Out;
	::gComm6D_OUT.Array[177] AT %QW."8YFLM01.0000.00I-1".EPL_FB_OUT_177_I2008_SB2Out;
	::gComm6D_OUT.Array[178] AT %QW."8YFLM01.0000.00I-1".EPL_FB_OUT_178_I2008_SB3Out;
	::gComm6D_OUT.Array[179] AT %QW."8YFLM01.0000.00I-1".EPL_FB_OUT_179_I2008_SB4Out;
	::gComm6D_OUT.Array[180] AT %QW."8YFLM01.0000.00I-1".EPL_FB_OUT_180_I2008_SB5Out;
	::gComm6D_OUT.Array[181] AT %QW."8YFLM01.0000.00I-1".EPL_FB_OUT_181_I2008_SB6Out;
	::gComm6D_OUT.Array[182] AT %QW."8YFLM01.0000.00I-1".EPL_FB_OUT_182_I2008_SB7Out;
	::gComm6D_OUT.Array[183] AT %QW."8YFLM01.0000.00I-1".EPL_FB_OUT_183_I2008_SB8Out;
	::gComm6D_OUT.Array[184] AT %QW."8YFLM01.0000.00I-1".EPL_FB_OUT_184_I2008_SB9Out;
	::gComm6D_OUT.Array[185] AT %QW."8YFLM01.0000.00I-1".EPL_FB_OUT_185_I2008_SBAOut;
	::gComm6D_OUT.Array[186] AT %QW."8YFLM01.0000.00I-1".EPL_FB_OUT_186_I2008_SBBOut;
	::gComm6D_OUT.Array[187] AT %QW."8YFLM01.0000.00I-1".EPL_FB_OUT_187_I2008_SBCOut;
	::gComm6D_OUT.Array[188] AT %QW."8YFLM01.0000.00I-1".EPL_FB_OUT_188_I2008_SBDOut;
	::gComm6D_OUT.Array[189] AT %QW."8YFLM01.0000.00I-1".EPL_FB_OUT_189_I2008_SBEOut;
	::gComm6D_OUT.Array[190] AT %QW."8YFLM01.0000.00I-1".EPL_FB_OUT_190_I2008_SBFOut;
	::gComm6D_OUT.Array[191] AT %QW."8YFLM01.0000.00I-1".EPL_FB_OUT_191_I2008_SC0Out;
	::gComm6D_OUT.Array[192] AT %QW."8YFLM01.0000.00I-1".EPL_FB_OUT_192_I2008_SC1Out;
	::gComm6D_OUT.Array[193] AT %QW."8YFLM01.0000.00I-1".EPL_FB_OUT_193_I2008_SC2Out;
	::gComm6D_OUT.Array[194] AT %QW."8YFLM01.0000.00I-1".EPL_FB_OUT_194_I2008_SC3Out;
	::gComm6D_OUT.Array[195] AT %QW."8YFLM01.0000.00I-1".EPL_FB_OUT_195_I2008_SC4Out;
	::gComm6D_OUT.Array[196] AT %QW."8YFLM01.0000.00I-1".EPL_FB_OUT_196_I2008_SC5Out;
	::gComm6D_OUT.Array[197] AT %QW."8YFLM01.0000.00I-1".EPL_FB_OUT_197_I2008_SC6Out;
	::gComm6D_OUT.Array[198] AT %QW."8YFLM01.0000.00I-1".EPL_FB_OUT_198_I2008_SC7Out;
	::gComm6D_OUT.Array[199] AT %QW."8YFLM01.0000.00I-1".EPL_FB_OUT_199_I2008_SC8Out;
END_VAR
```

### Config_1.assembly6d - 5APC2100_BY44_000/mapp6D/Config_1.assembly6d
```
Element gAssembly6D_1 (Type=assembly6d)
  Simulation6D = SimOff
  Shuttles:
    MaxShuttleCount = 4
    ShuttleIDMode = RealTimeID
    DefaultPosition:
      DefZ = 1.0
      DefRx = 0
      DefRy = 0
      DefRz = 0
    Limits:
      InPlaneLimits:
        InPlaneVelLim = 2
        InPlaneAccLim = 20
        InPlaneEmergDec = 20
      ShortAxLim:
        ShortAxAccLim:
          AccZLim = 10.0
          AccRxLim = 10.0
          AccRyLim = 10.0
          AccRzLim = 10.0
        ShortAxVelLim:
          VelZLim = 0.15
          VelRxLim = 0.1
          VelRyLim = 0.1
          VelRzLim = 0.3
  CyclicChannel6D:
    ReadChannel:
      Xaxis = TRUE
      Yaxis = TRUE
      Zaxis = TRUE
      Rxaxis = TRUE
      Ryaxis = TRUE
      Rzaxis = TRUE
  Fieldbus6D:
    SyncMode6D = ExternalPlkSync
    NodeNumber = 50
  IOMapp:
    Input = ::gComm6D_IN
    Output = ::gComm6D_OUT
  Layout:
    Layout6D[1] = Layout6D_1
```

## Logical view

Binary libraries used (declarations not repeated): operator, runtime, astime, AsIecCon, brsystem, AsBrStr, McAcp6D 1.01.0, McBase, brdkSTR, MTLookUp, sys_lib, standard

### Global.typ - Global data types
```iecst
TYPE
	Ctrl_typ : 	STRUCT
		Start : BOOL;
		Stop : BOOL;
		Reset : BOOL;
		Pause : BOOL;
	END_STRUCT;
	SysSettings_typ : 	STRUCT
		DemoType : BOOL; (*False = 2 segs true 4 segs*)
	END_STRUCT;
	Jog_typ : 	STRUCT
		Right : BOOL;
		Left : BOOL;
		Neg : BOOL;
		Pos : BOOL;
		ShuttleID : USINT;
		Degrees : REAL;
		ShortDistance : REAL;
		Distance : REAL;
		RyN : BOOL;
		RyP : BOOL;
		RxP : BOOL;
		RxN : BOOL;
		RzN : BOOL;
		RzP : BOOL;
		Down : BOOL;
		Up : BOOL;
		Zero : BOOL;
	END_STRUCT;
	Main_typ : 	STRUCT  (*Main control variable datatype*)
		Cmd : MainCmd_typ; (*Main commands*)
		Par : MainPar_typ; (*Main parameter*)
		Status : MainStatus_typ; (*Main status*)
	END_STRUCT;
	MainCmd_typ : 	STRUCT  (*Main commands type*)
		Power : BOOL; (*Power on the system*)
		Start : BOOL; (*Start a plane movement for the selected shuttle*)
		Pause : BOOL; (*Stop all shuttles in the system*)
		Resume : BOOL; (*Stop all shuttles in the system*)
		Stop : BOOL; (*Stop all shuttles in the system*)
		StopAll : BOOL; (*Stop all shuttles in the system*)
		Jog : Jog_typ;
		Land : BOOL;
		ResetAll : BOOL; (*Reset any active error*)
		ErrorReset : BOOL; (*Reset any active error*)
		Move6D : BOOL;
		Group : BOOL;
		Arc : BOOL;
		Weigh : BOOL;
		Tare : BOOL;
	END_STRUCT;
	MainPar_typ : 	STRUCT  (*Main parameter type*)
		SelectedIndex : UINT; (*Selected index in the global array of shuttle references*)
		JogShort : McAcp6DShortAxParType; (*Relevant motion parameter*)
		Jog : McAcp6DInPlaneParType; (*Relevant motion parameter*)
		Move6D : McAcp6DMove6DParType; (*Relevant motion parameter*)
		InPlane : McAcp6DInPlaneParType; (*Relevant motion parameter*)
		Arc : McAcp6DArcParType;
		ShortAxis : McAcp6DShortAx6DParType;
		ShrtVel : REAL;
		Accel : REAL;
		EndVelocity : REAL;
		Velocity : REAL;
	END_STRUCT;
	Position_typ : 	STRUCT
		X : REAL; (*mm*)
		Y : REAL; (*mm*)
		Z : REAL; (*mm*)
		Rx : REAL; (*Deg*)
		Ry : REAL; (*Deg*)
		Rz : REAL; (*Deg*)
		Payload : REAL; (*g*)
	END_STRUCT;
	MainStatus_typ : 	STRUCT  (*Main status type*)
		SelectedShuttleID : UINT; (*ID of the shuttle which was selected in the array*)
		AsmPlcOpenState : McAcp6dPLCopenStateEnum; (*PlcOpen state of the assembly*)
		ControllerState : McAcp6DControllerStateEnum; (*Current State of the ACOPOS 6D controller*)
		Disabled : BOOL; (*System is disabled*)
		Ready : BOOL; (*System is ready*)
		Homing : BOOL; (*System is homing*)
		Stopping : BOOL; (*System is stopping*)
		StartUp : BOOL; (*System is starting up*)
		ErrorStop : BOOL; (*System has an error*)
		ShuttlesPresent : USINT; (*Number of shuttles present*)
		ShtPresent : ARRAY[0..3]OF BOOL;
		Weight : ARRAY[0..3]OF REAL;
		Position : McAcp6DShPositionType;
	END_STRUCT;
	ShuttleStartup_typ : 	STRUCT
		initYPos : REAL;
		initXPos : REAL;
		nextStationSelector : STRING[80] := '0';
	END_STRUCT;
	MotorSegments_typ : 	STRUCT
		visible : BOOL := TRUE;
		ID : STRING[80];
	END_STRUCT;
	ShuttleReferenceArray_typ : 	STRUCT
		Reference : Mc6DShuttleType;
		ID : {REDUND_UNREPLICABLE} UINT;
	END_STRUCT;
	ShuttleInfo_typ : 	STRUCT
		ID : USINT;
		State : McAcp6DShStateEnum;
		Force : McAcp6DShForceType;
		Position : McAcp6DShPositionType;
		inUse : BOOL; (*DryStation Bool*)
	END_STRUCT;
	ShStatus_typ : 	STRUCT
		ShuttleInfo : ARRAY[0..MAX_NUM_SHUTTLES]OF ShuttleInfo_typ;
		ShuttleInfoVis : ARRAY[0..MAX_NUM_SHUTTLES]OF ShuttleInfo_typ;
	END_STRUCT;
END_TYPE
```

### Global.var - Global variables
```iecst
VAR
	gComm6D_IN : Mc6DControllerFBIOType; (*Communication var Input*)
	gComm6D_OUT : Mc6DControllerFBIOType; (*Communication var Output*)
END_VAR
(*CONSTANTS*)
VAR CONSTANT
	XY_MAX : REAL := 0.240;
	XY_MIN : REAL := 0.060;
	SEG_CENTER : REAL := 0.120;
	HALF_SHUTTLE : REAL := 0.06;
	MAX_INDEX_SHUTTLE : USINT := 4; (*Maximum index for a shuttles on the system (50 Shuttles)*)
	NR_OF_SEGMENTS : USINT := 9; (*10(0..9)*)
	MAX_NUM_SHUTTLES : USINT := 4; (*4 [0..3]*)
	NUM_SHUTTLES : USINT := 4; (*4[0.34]*)
	C_DISABLE : BOOL := FALSE;
	C_ENABLE : BOOL := TRUE;
	C_HIDE : BOOL := FALSE;
	C_SHOW : BOOL := TRUE;
END_VAR
(*Global Control Variable*)
VAR
	gMain : Main_typ; (*Global control variable*)
END_VAR
VAR RETAIN
	gSettings : SysSettings_typ;
END_VAR
VAR
	gShuttleReference : ARRAY[0..MAX_INDEX_SHUTTLE] OF ShuttleReferenceArray_typ; (*Global shuttle reference array*)
	gSegments : ARRAY[0..NR_OF_SEGMENTS] OF MotorSegments_typ;
	gShowMotorSegments : STRING[2000];
	gVisShuttle : ShStatus_typ;
	gShuttleStartupInfo : ARRAY[0..MAX_NUM_SHUTTLES] OF ShuttleStartup_typ;
	gCreateDemo : BOOL;
	gAssemblyY_max : REAL;
	gAssemblyX_max : REAL;
END_VAR
```


### Program Logical/MainCtrl (IEC)

#### Main.st - Init, cyclic, exit code
```iecst
PROGRAM _INIT

	visSelectedTab;

	IF gSettings.DemoType THEN
		gAssemblyX_max := (XY_MAX * 2)- HALF_SHUTTLE;
		gAssemblyY_max := (XY_MAX * 2)- HALF_SHUTTLE;
	ELSE
		gAssemblyX_max := (XY_MAX)- HALF_SHUTTLE;
		gAssemblyY_max := (XY_MAX * 2)- HALF_SHUTTLE;
	END_IF

	(* Initilaize communication *)
	gComm6D_IN;
	gComm6D_OUT;

	(* Initialize function blocks *)
	MC_BR_AsmReadStatus_Acp6D_0.Assembly    :=    ADR(gAssembly6D_1);
	MC_BR_AsmReadInfo_Acp6D_0.Assembly      :=    ADR(gAssembly6D_1);
	MC_BR_AsmPowerOn_Acp6D_0.Assembly       :=    ADR(gAssembly6D_1);
	MC_BR_AsmPowerOff_Acp6D_0.Assembly      :=    ADR(gAssembly6D_1);
	MC_BR_AsmGetShuttle_Acp6D_0.Assembly    :=    ADR(gAssembly6D_1);
	MC_BR_AsmStop_Acp6D_0.Assembly          :=    ADR(gAssembly6D_1);
	MC_BR_MoveInPlaneAsync_Acp6D_0.Assembly :=	  ADR(gAssembly6D_1);
	MC_BR_AsmGetInfo_Acp6D_0.Assembly 		:=	  ADR(gAssembly6D_1);

	(* Initialize main control variable *)
	(* InPlane Movement (X & Y) *)
	gMain.Par.InPlane.Acceleration          :=    20.0;   //[m/s²]
	gMain.Par.InPlane.Velocity              :=    2.0;    //[m/s]
	gMain.Par.InPlane.EndVelocity           :=    0.0;    //[m/s]
	// Top right position
	gMain.Par.InPlane.Position.X            :=    gAssemblyX_max; //[m]
	gMain.Par.InPlane.Position.Y            :=    gAssemblyY_max; //[m]
	gMain.Par.InPlane.Path                  :=    mcACP6D_PATH_X_THEN_Y;
	gMain.Par.InPlane.Mode                  :=    mcACP6D_MOVE_ABSOLUTE;

	(* Enable Diagnostic FUBs *)
	MC_BR_AsmReadStatus_Acp6D_0.Enable      :=    TRUE;
	MC_BR_AsmReadInfo_Acp6D_0.Enable        :=    TRUE;

	gMain.Cmd.Jog.Distance := 0.02;
	gMain.Cmd.Jog.Degrees := 0.5;

	gMain.Par.JogShort.Position.Rz := 0.5;
	gMain.Par.JogShort.Position.Ry := 0.0;
	gMain.Par.JogShort.Position.Rx := 0.0;
	gMain.Par.JogShort.Position.Z := 0.001;

	gMain.Par.JogShort.Velocity.Rx := 0.1;
	gMain.Par.JogShort.Velocity.Rz := 0.1;
	gMain.Par.JogShort.Velocity.Ry := 0.1;
	gMain.Par.JogShort.Velocity.Z := 0.005;

	gMain.Par.JogShort.Mode := mcACP6D_MOVE_ABSOLUTE;
	gMain.Par.JogShort.Rotation.Type := mcACP6D_SHORT_AX_ROT_ONLY;

	gMain.Par.JogShort.Rotation.Center.X := 60;
	gMain.Par.JogShort.Rotation.Center.Y := 60;

	gMain.Par.Jog.Velocity := 0.25;
	gMain.Par.Jog.Acceleration := 20;

	gMain.Par.Velocity := 2.0;
	gMain.Par.Accel := 20.0;

	zHeight[0] := 0.001;
	zHeight[1] := 0.004;
	zRollLimit[0] := 0.008;
	zRollLimit[1] := 0.055;

	MTLookUpTable_0.Enable := TRUE;
	MTLookUpTable_0.NodeVectorX := zHeight;
	MTLookUpTable_0.FcnValues := zRollLimit;
	MTLookUpTable_0.NumberOfNodes := 2;

END_PROGRAM

PROGRAM _CYCLIC

    (* Check for current status *)
	IF (gMain.Status.ErrorStop) THEN
		(* If an error occurs, go to the error state *)
		MainStep    :=    MAIN_ERROR;
	ELSIF (gMain.Status.StartUp) THEN
		(* As long, as the 6D - controller is in startup, stay in startup state *)
		MainStep    :=    MAIN_STARTUP;
	END_IF

	(* Limit the selected index for the shuttle array *)
	gMain.Par.SelectedIndex                                :=    LIMIT(0, gMain.Par.SelectedIndex, MIN(gMain.Status.ShuttlesPresent - 1, MAX_INDEX_SHUTTLE));
	(* State machine *)
	CASE MainStep OF

		MAIN_STARTUP:
			(* Wait for the 6D controller to be started *)
			IF (gMain.Status.Disabled) THEN
				(* If assembly is disabled *)
				MainStep                                :=    MAIN_DISABLED;
			ELSIF NOT(gMain.Status.StartUp) THEN
				(* If assembly is in any other state, disable it *)
				MainStep                                :=    MAIN_POWER_OFF;
			END_IF

		MAIN_POWER_OFF:
			(* Activate Function block *)
			MC_BR_AsmPowerOff_Acp6D_0.Execute            :=    TRUE;
			(* Wait for the command to be done *)
			IF (MC_BR_AsmPowerOff_Acp6D_0.Done) THEN
				(* Reset the function block *)
				MC_BR_AsmPowerOff_Acp6D_0.Execute        :=    FALSE;
				(* Next step *)
				MainStep                                :=    MAIN_DISABLED;
			ELSIF (MC_BR_AsmPowerOff_Acp6D_0.Error) THEN
				(* Next step *)
				MainStep                                :=    MAIN_ERROR;
			END_IF

		MAIN_DISABLED:
			IF (gMain.Cmd.Power) THEN
				(* Next step *)
				MainStep                                :=    MAIN_POWER_ON;
			END_IF

		MAIN_POWER_ON:
			(* Activate Function block *)
			MC_BR_AsmPowerOn_Acp6D_0.Execute            :=    TRUE;
			(* Wait for the command to be done *)
			IF (MC_BR_AsmPowerOn_Acp6D_0.Done) THEN
				(* Reset the function block *)
				MC_BR_AsmPowerOn_Acp6D_0.Execute        :=    FALSE;
				(* Delete data from global shuttle array *)
				brsmemset(ADR(gShuttleReference),0,SIZEOF(gShuttleReference));
				(* Next step *)
				MainStep                                :=    MAIN_GET_SHUTTLE;
			ELSIF (MC_BR_AsmPowerOn_Acp6D_0.Error) THEN
				(* Next step *)
				MainStep                                :=    MAIN_ERROR;
			END_IF

		MAIN_GET_SHUTTLE:
			(* Enable the function block *)
			MC_BR_AsmGetShuttle_Acp6D_0.Enable            :=    TRUE;
			(* Wait until the data is valid *)
			IF (MC_BR_AsmGetShuttle_Acp6D_0.Valid) THEN
				(* Check any shuttle is present *)
				IF (MC_BR_AsmGetShuttle_Acp6D_0.TotalCount > 0) THEN
					(* Reset the "next" command *)
					MC_BR_AsmGetShuttle_Acp6D_0.Next    :=    FALSE;
					(* Save the number of shuttles *)
					gMain.Status.ShuttlesPresent        :=    UINT_TO_USINT(MC_BR_AsmGetShuttle_Acp6D_0.TotalCount);
					(* Next step *)
					MainStep                            :=    MAIN_GET_SHUTTLE_WAIT;
				ELSE
					(* No shuttles present *)
					gMain.Status.ShuttlesPresent        :=    0;
					(* Disable the function block *)
					MC_BR_AsmGetShuttle_Acp6D_0.Enable  :=    TRUE;
					(* Next step *)
					MainStep                            :=    MAIN_READY;
				END_IF
			END_IF

		MAIN_GET_SHUTTLE_WAIT:
			(* Search for the next free index *)
			FOR i := 0 TO MAX_INDEX_SHUTTLE DO
				IF (gShuttleReference[i].ID = 0) THEN
					(* Save the current array index and exit the loop *)
					NextFreeIndex                        :=    i;
					EXIT;
				END_IF
			END_FOR
			(* Save the shuttle reference *)
			gShuttleReference[NextFreeIndex].Reference    :=   MC_BR_AsmGetShuttle_Acp6D_0.Shuttle;
			gShuttleReference[NextFreeIndex].ID           :=   MC_BR_AsmGetShuttle_Acp6D_0.AdditionalInfo.ShuttleID;
			(* Check if there are more shuttles to read out *)
			IF (MC_BR_AsmGetShuttle_Acp6D_0.RemainingCount > 0) THEN
				(* Get next shuttle *)
				MC_BR_AsmGetShuttle_Acp6D_0.Next        :=    TRUE;
				(* Next step *)
				MainStep                                :=    MAIN_GET_SHUTTLE;
			ELSE
				(* Reset the function block *)
				MC_BR_AsmGetShuttle_Acp6D_0.Enable      :=    FALSE;
				(* Next step *)
				MainStep                                :=    MAIN_READY;
			END_IF

		MAIN_READY:

			visShowReset := C_HIDE;

			IF NOT(gMain.Cmd.Power) OR (gMain.Status.Disabled) THEN
				(* Power off the system, if the power command is reset, or the assembly is disabled *)
				(* Reset command *)
				gMain.Cmd.Power                         :=    FALSE;
				(* Next step *)
				MainStep                                :=    MAIN_POWER_OFF;
			ELSIF (gMain.Cmd.Start) THEN
				(* Start a movement when the command is set and a valid shuttleID is selected *)
				(* Reset command *)
				gMain.Cmd.Start                         :=    FALSE;
				(* Next step *)
				MainStep                                :=    MAIN_START_MOVEMENT;
			ELSIF (gMain.Cmd.StopAll) THEN
				(* Stop all shuttles in the assembly, if the command is set *)
				(* Reset command *)
				gMain.Cmd.StopAll                       :=    FALSE;
				(* Next step *)
				MainStep                                :=    MAIN_STOP_ALL_SHUTTLES;
			ELSIF gMain.Cmd.Land THEN
				gMain.Cmd.Land := FALSE;
				MainStep  								:=    MAIN_LEVITATE;
			ELSIF gMain.Cmd.Move6D THEN
				gMain.Cmd.Move6D := FALSE;
				MainStep                                :=    MAIN_MOVE_6D;
			ELSIF gMain.Cmd.Arc THEN
				gMain.Cmd.Arc := FALSE;
				MainStep                                :=    MAIN_MOVE_ARC;
			ELSIF gMain.Cmd.Group THEN
				gMain.Cmd.Group := FALSE;
				MainStep                                :=    MAIN_MOVE_GROUP;
			ELSIF gMain.Cmd.Weigh THEN
				gMain.Cmd.Weigh := FALSE;
				MainStep                                :=    MAIN_WEIGH;
			ELSIF gMain.Cmd.Pause THEN
				gMain.Cmd.Pause := FALSE;
				MainStep  								:=    MAIN_HALT_SELECTED;
			ELSIF gMain.Cmd.Resume THEN
				gMain.Cmd.Resume := FALSE;
				MainStep  								:=    MAIN_RESUME_SELECTED;
			ELSIF gMain.Cmd.Stop THEN
				gMain.Cmd.Stop := FALSE;
				MainStep  								:=    MAIN_STOP_SELECTED;
			ELSIF gMain.Cmd.ResetAll THEN
				gMain.Cmd.ResetAll := FALSE;
				MainStep  								:=    MAIN_RECOVER_ALL; // Recover disabled shuttles
			END_IF

			// Jog command recieved
			IF EDGEPOS(gMain.Cmd.Jog.Left OR gMain.Cmd.Jog.Right OR gMain.Cmd.Jog.Neg OR gMain.Cmd.Jog.Pos OR gMain.Cmd.Jog.RzP OR gMain.Cmd.Jog.RzN OR gMain.Cmd.Jog.RxP OR gMain.Cmd.Jog.RxN OR gMain.Cmd.Jog.RyP OR gMain.Cmd.Jog.RyN OR gMain.Cmd.Jog.Up OR gMain.Cmd.Jog.Down)OR(gMain.Cmd.Jog.Zero)THEN
				MainStep             :=    MAIN_JOG_SHUTTLE;
			END_IF

		MAIN_WEIGH:

			WeighAct;

		MAIN_START_MOVEMENT:

			(* Activate the function block *)
			MC_BR_MoveInPlane_Acp6D_0.Shuttle            :=    ADR(gShuttleReference[gMain.Par.SelectedIndex].Reference);
			MC_BR_MoveInPlane_Acp6D_0.Parameters        :=    gMain.Par.InPlane; //Parameter set in INIT, can be modified in Watch
			MC_BR_MoveInPlane_Acp6D_0.Execute            :=    TRUE;
			(* Wait for the command to be accepted *)
			IF (MC_BR_MoveInPlane_Acp6D_0.Acknowledge) THEN
				(* Reset the function block *)
				MC_BR_MoveInPlane_Acp6D_0.Execute        :=    FALSE;
				(* Next step *)
				MainStep                                :=    MAIN_READY;
			ELSIF (MC_BR_MoveInPlane_Acp6D_0.Error) THEN
				(* Next step *)
				MainStep                                :=    MAIN_ERROR;
			END_IF

		MAIN_JOG_SHUTTLE:

			// Jog function
			JogAct;

			TON_0.PT := t#1s;
			TON_0.IN := NOT(gMain.Cmd.Jog.Left OR gMain.Cmd.Jog.Right OR gMain.Cmd.Jog.Neg OR gMain.Cmd.Jog.Pos OR gMain.Cmd.Jog.RxP OR gMain.Cmd.Jog.RxN OR gMain.Cmd.Jog.RyP OR gMain.Cmd.Jog.RyN OR gMain.Cmd.Jog.Up OR gMain.Cmd.Jog.Down);

			IF TON_0.Q THEN
				TON_0.IN := FALSE;
				MainStep := MAIN_READY;
				MC_BR_ShStop_Acp6D_0.Execute := FALSE;
			END_IF

		MAIN_LEVITATE:

			MC_BR_ShLevitation_Acp6D_0.Shuttle := ADR(gShuttleReference[gMain.Par.SelectedIndex].Reference);

			IF(gVisShuttle.ShuttleInfoVis[gMain.Par.SelectedIndex].State <> mcACP6D_SH_STATE_LANDED)THEN
				MC_BR_ShLevitation_Acp6D_0.Parameters.Level := mcACP6D_LEVEL_LAND;
				MC_BR_ShLevitation_Acp6D_0.Execute := TRUE;
			ELSE
				MC_BR_ShLevitation_Acp6D_0.Parameters.Level := mcACP6D_LEVEL_LEVITATE;
				MC_BR_ShLevitation_Acp6D_0.Execute := TRUE;
			END_IF

			IF MC_BR_ShLevitation_Acp6D_0.Done THEN
				(* Next step *)
				MC_BR_ShLevitation_Acp6D_0.Execute := FALSE;
				MainStep                           := MAIN_READY;
			ELSIF MC_BR_ShLevitation_Acp6D_0.Error THEN
				(* Next step *)
				ErrorStep := MainStep;
				ErrorNumber := MC_BR_ShLevitation_Acp6D_0.ErrorID;
				MC_BR_ShLevitation_Acp6D_0.Execute := FALSE;
				MainStep                           := MAIN_ERROR;
			END_IF

		MAIN_MOVE_6D:

			gMain.Par.Arc.Option := mcACP6D_ARC_ANGULAR;

			MC_BR_Move6D_Acp6D_0.Shuttle := ADR(gShuttleReference[gMain.Par.SelectedIndex].Reference);
			MC_BR_Move6D_Acp6D_0.Execute := TRUE;

			gMain.Par.Move6D.InPlane.Velocity := gMain.Par.Velocity;
			gMain.Par.Move6D.InPlane.Acceleration := gMain.Par.Accel;

			MC_BR_Move6D_Acp6D_0.Parameters := gMain.Par.Move6D;
			MC_BR_Move6D_Acp6D_0.Parameters.InPlane.Position.X := gMain.Par.Move6D.InPlane.Position.X/1000; // convert to m
			MC_BR_Move6D_Acp6D_0.Parameters.InPlane.Position.Y := gMain.Par.Move6D.InPlane.Position.Y/1000; // convert to m
			MC_BR_Move6D_Acp6D_0.Parameters.ShortAxis.Position.Z := gMain.Par.Move6D.ShortAxis.Position.Z/1000; // convert to m
			MC_BR_Move6D_Acp6D_0.Parameters.ShortAxis.Position.Rx := gMain.Par.Move6D.ShortAxis.Position.Rx * 0.017453293; // convert to mrad
			MC_BR_Move6D_Acp6D_0.Parameters.ShortAxis.Position.Ry := gMain.Par.Move6D.ShortAxis.Position.Ry * 0.017453293; // convert to mrad
			MC_BR_Move6D_Acp6D_0.Parameters.ShortAxis.Position.Rz := gMain.Par.Move6D.ShortAxis.Position.Rz * 0.017453293; // convert to mrad

			MC_BR_Move6D_Acp6D_0.CommandLabel := 150;

			IF MC_BR_Move6D_Acp6D_0.Done OR MC_BR_Move6D_Acp6D_0.Acknowledge THEN
				MC_BR_Move6D_Acp6D_0.Execute := FALSE;
				MainStep          := MAIN_READY;
			ELSIF MC_BR_Move6D_Acp6D_0.Error THEN
				ErrorStep := MainStep;
				ErrorNumber := MC_BR_Move6D_Acp6D_0.ErrorID;
				MC_BR_MoveArc_Acp6D_0.Execute := FALSE;
				MainStep          := MAIN_ERROR;
			END_IF

		MAIN_MOVE_ARC:

			gMain.Par.Arc.Option := mcACP6D_ARC_ANGULAR;

			MC_BR_MoveArc_Acp6D_0.Shuttle := ADR(gShuttleReference[gMain.Par.SelectedIndex].Reference);
			MC_BR_MoveArc_Acp6D_0.Execute := TRUE;

			gMain.Par.Arc.Velocity := gMain.Par.Velocity;
			gMain.Par.Arc.Acceleration := gMain.Par.Accel;
			gMain.Par.Arc.EndVelocity := gMain.Par.EndVelocity;

			MC_BR_MoveArc_Acp6D_0.Parameters := gMain.Par.Arc;
			MC_BR_MoveArc_Acp6D_0.Parameters.Angular.Angle := gMain.Par.Arc.Angular.Angle * 0.017453293; // convert to mrad
			MC_BR_MoveArc_Acp6D_0.Parameters.Angular.Center.X := gMain.Par.Arc.Angular.Center.X/1000; // convert to m
			MC_BR_MoveArc_Acp6D_0.Parameters.Angular.Center.Y := gMain.Par.Arc.Angular.Center.Y/1000;
			MC_BR_MoveArc_Acp6D_0.CommandLabel := 160;

			IF MC_BR_MoveArc_Acp6D_0.Done OR MC_BR_MoveArc_Acp6D_0.Acknowledge THEN
				MC_BR_MoveArc_Acp6D_0.Execute := FALSE;
				MainStep          := MAIN_READY;
			ELSIF MC_BR_MoveArc_Acp6D_0.Error THEN
				ErrorStep := MainStep;
				ErrorNumber := MC_BR_MoveArc_Acp6D_0.ErrorID;
				MC_BR_MoveArc_Acp6D_0.Execute := FALSE;
				MainStep          := MAIN_ERROR;
			END_IF

		MAIN_MOVE_GROUP:

		MAIN_RECOVER:

			IF(gVisShuttle.ShuttleInfoVis[gMain.Par.SelectedIndex].State = mcACP6D_SH_STATE_DISABLED)THEN
				MC_BR_ShRecover_Acp6D_0.Shuttle := ADR(gShuttleReference[gMain.Par.SelectedIndex].Reference);
				MC_BR_ShRecover_Acp6D_0.Execute := TRUE;
			END_IF

			IF MC_BR_ShRecover_Acp6D_0.Done THEN
				MC_BR_ShRecover_Acp6D_0.Execute := FALSE;
				MainStep          := MAIN_READY;
			ELSIF MC_BR_ShRecover_Acp6D_0.Error THEN
				ErrorStep := MainStep;
				ErrorNumber := MC_BR_ShRecover_Acp6D_0.ErrorID;
				MC_BR_ShRecover_Acp6D_0.Execute := FALSE;
				MainStep          := MAIN_ERROR;
			END_IF

		MAIN_RECOVER_ALL:

			IF (k <=(gMain.Status.ShuttlesPresent - 1))THEN
				MC_BR_ShRecover_Acp6D_0.Shuttle := ADR(gShuttleReference[k].Reference);
				IF ((gVisShuttle.ShuttleInfoVis[k].State = mcACP6D_SH_STATE_DISABLED)) THEN
					MC_BR_ShRecover_Acp6D_0.Execute := TRUE;
				ELSIF(k < gMain.Status.ShuttlesPresent)THEN
					k := k+1;
				END_IF

				IF MC_BR_ShRecover_Acp6D_0.Done THEN
					k := k+1;
					MC_BR_ShRecover_Acp6D_0.Execute := FALSE;
					IF (k = gMain.Status.ShuttlesPresent) THEN
						k := 0;
						MainStep          := MAIN_READY;
						visResetSelected := C_HIDE;
					END_IF
				ELSIF MC_BR_ShRecover_Acp6D_0.Error THEN
					ErrorStep := MainStep;
					ErrorNumber := MC_BR_ShRecover_Acp6D_0.ErrorID;
					MC_BR_ShRecover_Acp6D_0.Execute := FALSE;
					k := 0;
					MainStep          := MAIN_ERROR;
					visResetSelected := C_HIDE;

				END_IF
			ELSE
				k := 0;
				MainStep          := MAIN_READY;
					visResetSelected := C_HIDE;
			END_IF

		MAIN_HALT_SELECTED:

				MC_BR_ShHalt_Acp6D_0.Shuttle := ADR(gShuttleReference[gMain.Par.SelectedIndex].Reference);
				MC_BR_ShHalt_Acp6D_0.Option := mcACP6D_HALT;
				MC_BR_ShHalt_Acp6D_0.Execute := TRUE;

			IF MC_BR_ShHalt_Acp6D_0.Done THEN
				MC_BR_ShHalt_Acp6D_0.Execute := FALSE;
				MainStep          := MAIN_READY;
			ELSIF MC_BR_ShHalt_Acp6D_0.Error THEN
				ErrorStep := MainStep;
				ErrorNumber := MC_BR_ShHalt_Acp6D_0.ErrorID;
				MC_BR_ShHalt_Acp6D_0.Execute := FALSE;
				MainStep          := MAIN_ERROR;
			END_IF

		MAIN_RESUME_SELECTED:

			MC_BR_ShHalt_Acp6D_0.Shuttle := ADR(gShuttleReference[gMain.Par.SelectedIndex].Reference);
			MC_BR_ShHalt_Acp6D_0.Option := mcACP6D_CONTINUE;
			MC_BR_ShHalt_Acp6D_0.Execute := TRUE;

			IF MC_BR_ShHalt_Acp6D_0.Done THEN
				MC_BR_ShHalt_Acp6D_0.Execute := FALSE;
				MainStep          := MAIN_READY;
			ELSIF MC_BR_ShHalt_Acp6D_0.Error THEN
				ErrorStep := MainStep;
				ErrorNumber := MC_BR_ShHalt_Acp6D_0.ErrorID;
				MC_BR_ShHalt_Acp6D_0.Execute := FALSE;
				MainStep          := MAIN_ERROR;
			END_IF

		MAIN_STOP_SELECTED:

				MC_BR_ShStop_Acp6D_0.Shuttle := ADR(gShuttleReference[gMain.Par.SelectedIndex].Reference);
				MC_BR_ShStop_Acp6D_0.Execute := TRUE;

			IF MC_BR_ShStop_Acp6D_0.Done OR(gVisShuttle.ShuttleInfoVis[gMain.Par.SelectedIndex].State = mcACP6D_SH_STATE_IDLING)THEN
				MC_BR_ShStop_Acp6D_0.Execute := FALSE;
				MainStep          := MAIN_READY;
			ELSIF MC_BR_ShStop_Acp6D_0.Error THEN
				ErrorStep := MainStep;
				ErrorNumber := MC_BR_ShStop_Acp6D_0.ErrorID;
				MC_BR_ShStop_Acp6D_0.Execute := FALSE;
				MainStep          := MAIN_ERROR;
			END_IF

		MAIN_STOP_ALL_SHUTTLES:
			(* Activate Function block *)
			MC_BR_AsmStop_Acp6D_0.Execute               :=    TRUE;
			(* Wait for the command to be done *)
			IF (MC_BR_AsmStop_Acp6D_0.Done) THEN
				(* Reset the function block *)
				MC_BR_AsmStop_Acp6D_0.Execute           :=    FALSE;
				(* Next step *)
				MainStep                                :=    MAIN_READY;
			ELSIF (MC_BR_AsmStop_Acp6D_0.Error) THEN
				(* Next step *)
				ErrorStep := MainStep;
				ErrorNumber := MC_BR_AsmStop_Acp6D_0.ErrorID;
				MainStep                                :=    MAIN_ERROR;
			END_IF

		MAIN_ERROR:
			visShowReset := C_SHOW;
			(* Reset the assembly after diagnosis *)
			IF (gMain.Cmd.ErrorReset) AND NOT(gMain.Status.ErrorStop) THEN
				(* Reset command *)
				gMain.Cmd.ErrorReset                    :=    FALSE;
				(* Reset function blocks *)
				MC_BR_AsmPowerOn_Acp6D_0.Execute        :=    FALSE;
				MC_BR_AsmPowerOff_Acp6D_0.Execute       :=    FALSE;
				MC_BR_AsmGetShuttle_Acp6D_0.Enable      :=    FALSE;
				MC_BR_AsmGetShuttle_Acp6D_0.Next        :=    FALSE;
				MC_BR_AsmStop_Acp6D_0.Execute           :=    FALSE;
				MC_BR_MoveInPlane_Acp6D_0.Execute       :=    FALSE;

				// Reset Commands
				gMain.Cmd.Arc                         	:=    FALSE;
				gMain.Cmd.Stop                         	:=    FALSE;
				gMain.Cmd.Move6D                       	:=    FALSE;
				gMain.Cmd.Weigh                        	:=    FALSE;
				gMain.Cmd.StopAll                      	:=    FALSE;
				gMain.Cmd.Land                         	:=    FALSE;

				ErrorNumber := 0;

				(* Next step *)
				IF (gMain.Status.Disabled) THEN
					(* Reset command *)
					gMain.Cmd.Power                     :=    FALSE;
					MainStep                            :=    MAIN_DISABLED;
				ELSIF (gMain.Status.Ready) THEN
					(* Reset command *)
					gMain.Cmd.Power                     :=    TRUE;
					MainStep                            :=    MAIN_READY;
				END_IF
			END_IF
	END_CASE

	statusCount := 0;
	FOR i := 0 TO (NUM_SHUTTLES-1) DO

		MC_BR_ShReadInfo_Acp6D_0[i].Shuttle					:= ADR(gShuttleReference[i].Reference);
		MC_BR_ShReadInfo_Acp6D_0[i].Enable					:= gMain.Status.Ready; //gAcp6DCtrl.Status.PowerOn;

		MC_BR_ReadCyclicPosition_Acp6D_0[i].Shuttle 		:= ADR(gShuttleReference[i].Reference);;
		MC_BR_ReadCyclicPosition_Acp6D_0[i].Enable			:= gMain.Status.Ready; //gAcp6DCtrl.Status.PowerOn;

		IF(MC_BR_ShReadInfo_Acp6D_0[i].Valid)THEN

			gVisShuttle.ShuttleInfo[i].Position 	:= MC_BR_ShReadInfo_Acp6D_0[i].ShuttleInfo.Position;
			gVisShuttle.ShuttleInfo[i].ID			:= UINT_TO_USINT(MC_BR_ShReadInfo_Acp6D_0[i].ShuttleInfo.ShuttleID);
			gVisShuttle.ShuttleInfo[i].State		:= MC_BR_ShReadInfo_Acp6D_0[i].ShuttleInfo.State;

			gVisShuttle.ShuttleInfoVis[i].State	:= MC_BR_ShReadInfo_Acp6D_0[i].ShuttleInfo.State;
			gVisShuttle.ShuttleInfoVis[i].Position.X := gVisShuttle.ShuttleInfo[i].Position.X* 1000.0;
			gVisShuttle.ShuttleInfoVis[i].Position.Y := gVisShuttle.ShuttleInfo[i].Position.Y* 1000.0;
			gVisShuttle.ShuttleInfoVis[i].Position.Z := gVisShuttle.ShuttleInfo[i].Position.Z* 1000.0;
			gVisShuttle.ShuttleInfoVis[i].Position.Rx := gVisShuttle.ShuttleInfo[i].Position.Rx* 1000.0;
			gVisShuttle.ShuttleInfoVis[i].Position.Ry := gVisShuttle.ShuttleInfo[i].Position.Ry* 1000.0;
			gVisShuttle.ShuttleInfoVis[i].Position.Rz := gVisShuttle.ShuttleInfo[i].Position.Rz* 1000.0;
			gVisShuttle.ShuttleInfoVis[i].ID := gVisShuttle.ShuttleInfo[i].ID;

		ELSIF MC_BR_ShReadInfo_Acp6D_0[i].Error OR MC_BR_ShReadInfo_Acp6D_0[i].Error THEN

			MC_BR_ShReadInfo_Acp6D_0[i].Enable 			:= FALSE;
			MC_BR_ReadCyclicPosition_Acp6D_0[i].Enable	:= FALSE;

		END_IF

		IF ((gVisShuttle.ShuttleInfoVis[i].State = mcACP6D_SH_STATE_DISABLED)) THEN
			statusCount := statusCount + 1;
		END_IF

		IF statusCount > 0 THEN
			visResetSelected := C_SHOW;
		ELSE
			visResetSelected := C_HIDE;
			statusCount := 0;
		END_IF

		MC_BR_ShReadInfo_Acp6D_0[i]();
		MC_BR_ReadCyclicPosition_Acp6D_0[i]();

	END_FOR

	// Set present Flags for visability
	IF gMain.Status.ShuttlesPresent > 0 THEN
		FOR i:= 0 TO (gMain.Status.ShuttlesPresent - 1) DO
			gMain.Status.ShtPresent[i] := TRUE;
		END_FOR
	END_IF

	// Change the Land and take off image
	IF(gVisShuttle.ShuttleInfoVis[gMain.Par.SelectedIndex].State <> mcACP6D_SH_STATE_LANDED)THEN
		visuLandText := 'Media/Land.png';
	ELSE
		visuLandText := 'Media/Levitate.png';
	END_IF

	// read assembly info or clear error

	IF MC_BR_AsmGetInfo_Acp6D_0.Error THEN
		MC_BR_AsmGetInfo_Acp6D_0.Execute := FALSE;
	ELSE
		MC_BR_AsmGetInfo_Acp6D_0.Execute 		:= gMain.Status.Ready;
	END_IF

	(* Call Function blocks *)
	MC_BR_AsmReadStatus_Acp6D_0();
	MC_BR_AsmReadInfo_Acp6D_0();
	MC_BR_AsmPowerOn_Acp6D_0();
	MC_BR_AsmPowerOff_Acp6D_0();
	MC_BR_AsmGetShuttle_Acp6D_0();
	MC_BR_AsmStop_Acp6D_0();
	MC_BR_MoveInPlane_Acp6D_0();
	MC_BR_MoveShortAxis_Acp6D_0();
	MC_BR_ShStop_Acp6D_0();
	MC_BR_ShLevitation_Acp6D_0();
	MC_BR_MoveInPlaneAsync_Acp6D_0();
	MC_BR_ShGetPayload_Acp6D_0();
	MC_BR_Move6D_Acp6D_0();
	MC_BR_MoveArc_Acp6D_0();
	MC_BR_ShRecover_Acp6D_0();
	MC_BR_ShHalt_Acp6D_0();
	MC_BR_AsmGetInfo_Acp6D_0();

	MTLookUpTable_0();
	TON_0();

	(* Assign Current Info and Status of the Assembly *)
	gMain.Status.AsmPlcOpenState        :=    MC_BR_AsmReadInfo_Acp6D_0.AssemblyInfo.AssemblyState;
	gMain.Status.ControllerState        :=    MC_BR_AsmReadInfo_Acp6D_0.AssemblyInfo.Controller6DState;
	gMain.Status.StartUp                :=    MC_BR_AsmReadStatus_Acp6D_0.AssemblyStartUp;
	gMain.Status.Disabled               :=    MC_BR_AsmReadStatus_Acp6D_0.AssemblyDisabled;
	gMain.Status.Homing                 :=    MC_BR_AsmReadStatus_Acp6D_0.AssemblyHoming;
	gMain.Status.Ready                  :=    MC_BR_AsmReadStatus_Acp6D_0.AssemblyReady;
	gMain.Status.Stopping               :=    MC_BR_AsmReadStatus_Acp6D_0.AssemblyStopping;
	gMain.Status.ErrorStop              :=    MC_BR_AsmReadStatus_Acp6D_0.AssemblyErrorStop;

	// Display the ^D Status Text
	CASE gMain.Status.AsmPlcOpenState OF
		mcACP6D_DISABLED:
			visStatusText := 'Disabled';
			visPowerImage := 'Media/Power.png';
		mcACP6D_HOMING:
			visStatusText := 'Homeing';
			visPowerImage := 'Media/PowerHome.png';
		mcACP6D_READY:
			visStatusText := 'Running';
			visPowerImage := 'Media/PowerOn.png';
		mcACP6D_STOPPING:
			visStatusText := 'Stopping';
			visPowerImage := 'Media/PowerStop.png';
		mcACP6D_ERRORSTOP:
			visStatusText := 'Error Stop';
			visPowerImage := 'Media/PowerRed.png';
		mcACP6D_STARTUP:
			visStatusText := 'Starting Up';
			visPowerImage := 'Media/PowerStarting.png';
		mcACP6D_INVALID_CONFIGURATION:
			visStatusText := 'Problem with Config';
			visPowerImage := 'Media/PowerConfig.png';
	END_CASE

	// Create the demo macro when first going to demo tab
	IF EDGEPOS(visSelectedTab = 4)AND(gMain.Status.ShuttlesPresent > 0)THEN
		gCreateDemo := TRUE;
	END_IF

	(* Show the ID of the currently selected shuttle reference *)
	gMain.Status.SelectedShuttleID      :=    gShuttleReference[gMain.Par.SelectedIndex].ID;
	gMain.Status.Position 				:=	  gVisShuttle.ShuttleInfoVis[gMain.Par.SelectedIndex].Position;
	gMain.Status.Position.Rx := gVisShuttle.ShuttleInfoVis[gMain.Par.SelectedIndex].Position.Rx / 17.453293;
	gMain.Status.Position.Ry := gVisShuttle.ShuttleInfoVis[gMain.Par.SelectedIndex].Position.Ry / 17.453293;
	gMain.Status.Position.Rz := gVisShuttle.ShuttleInfoVis[gMain.Par.SelectedIndex].Position.Rz / 17.453293;

END_PROGRAM

PROGRAM _EXIT
    (* Disable FUBs *)
	MC_BR_AsmReadStatus_Acp6D_0.Enable    :=    TRUE;
	MC_BR_AsmReadInfo_Acp6D_0.Enable    :=    TRUE;

	(* Call Function blocks *)
	MC_BR_AsmReadStatus_Acp6D_0();
	MC_BR_AsmReadInfo_Acp6D_0();
END_PROGRAM
```

#### Types.typ - Local data types
```iecst
TYPE
	MainStep_enum :
		( (*States for the main state machine*)
		MAIN_STARTUP,
		MAIN_POWER_OFF,
		MAIN_DISABLED,
		MAIN_POWER_ON,
		MAIN_GET_SHUTTLE,
		MAIN_GET_SHUTTLE_WAIT,
		MAIN_READY,
		MAIN_START_MOVEMENT,
		MAIN_JOG_SHUTTLE,
		MAIN_WEIGH,
		MAIN_MOVE_6D,
		MAIN_MOVE_ARC,
		MAIN_MOVE_GROUP,
		MAIN_LEVITATE,
		MAIN_HALT_SELECTED,
		MAIN_RESUME_SELECTED,
		MAIN_STOP_SELECTED,
		MAIN_STOP_ALL_SHUTTLES,
		MAIN_RECOVER_ALL,
		MAIN_RECOVER,
		MAIN_ERROR
		);
END_TYPE
```

#### Variables.var - Local variables
```iecst
VAR
	MainStep : MainStep_enum; (*Variable for the state machine*)
END_VAR
(*Function Blocks*)
VAR
	MC_BR_AsmReadStatus_Acp6D_0 : MC_BR_AsmReadStatus_Acp6D;
	MC_BR_AsmReadInfo_Acp6D_0 : MC_BR_AsmReadInfo_Acp6D;
	MC_BR_AsmPowerOn_Acp6D_0 : MC_BR_AsmPowerOn_Acp6D;
	MC_BR_AsmPowerOff_Acp6D_0 : MC_BR_AsmPowerOff_Acp6D;
	MC_BR_AsmGetShuttle_Acp6D_0 : MC_BR_AsmGetShuttle_Acp6D;
	MC_BR_AsmStop_Acp6D_0 : MC_BR_AsmStop_Acp6D;
	MC_BR_MoveInPlane_Acp6D_0 : MC_BR_MoveInPlane_Acp6D;
	MTLookUpTable_0 : MTLookUpTable;
	MC_BR_ShLevitation_Acp6D_0 : MC_BR_ShLevitation_Acp6D;
	MC_BR_MoveInPlaneAsync_Acp6D_0 : MC_BR_MoveInPlaneAsync_Acp6D;
	MC_BR_ShGetPayload_Acp6D_0 : MC_BR_ShGetPayload_Acp6D;
	MC_BR_ShReadInfo_Acp6D_0 : ARRAY[0..MAX_NUM_SHUTTLES] OF MC_BR_ShReadInfo_Acp6D;
	MC_BR_ReadCyclicPosition_Acp6D_0 : ARRAY[0..MAX_NUM_SHUTTLES] OF MC_BR_ReadCyclicPosition_Acp6D;
	MC_BR_ShStop_Acp6D_0 : MC_BR_ShStop_Acp6D;
	MC_BR_MoveShortAxis_Acp6D_0 : MC_BR_MoveShortAxis_Acp6D;
	MC_BR_Move6D_Acp6D_0 : MC_BR_Move6D_Acp6D;
	MC_BR_MoveArc_Acp6D_0 : MC_BR_MoveArc_Acp6D;
	MC_BR_ShRecover_Acp6D_0 : MC_BR_ShRecover_Acp6D;
	MC_BR_ShHalt_Acp6D_0 : MC_BR_ShHalt_Acp6D;
	TON_0 : TON;
END_VAR
(*Local Vars*)
VAR
	NextFreeIndex : USINT; (*Next free index in the global shuttle array*)
	TareWeight : ARRAY[0..3] OF REAL;
	YawLimit : REAL;
	zHeight : ARRAY[0..49] OF REAL;
	zRollLimit : ARRAY[0..49] OF REAL;
END_VAR
(*Visualisation status/visability links*)
VAR
	visuLandText : STRING[80];
	visStatusText : STRING[80];
	visPowerImage : STRING[80];
	visResetSelected : BOOL;
	visSelectedTab : UINT;
END_VAR
(*State machine states*)
VAR
	stateWeigh : UDINT;
	statePMT : UDINT;
END_VAR
(*Counters*)
VAR
	i : USINT;
	j : USINT;
	k : UINT;
	statusCount : USINT;
	MC_BR_AsmGetInfo_Acp6D_0 : MC_BR_AsmGetInfo_Acp6D;
	visShowReset : BOOL;
	ErrorStep : MainStep_enum;
	ErrorNumber : DINT;
	AverageWeightShtSum : ARRAY[0..3] OF REAL;
	AverageWeightShtl : ARRAY[0..3,0..499] OF REAL;
	AverageWeightShtlSum : ARRAY[0..3] OF REAL;
	l : UINT;
	m : UINT;
END_VAR
```

#### JogAct.st
```iecst
ACTION JogAct:

	// Get the position of the sleected shuttle
	gMain.Par.Jog.Position.X := (gVisShuttle.ShuttleInfo[gMain.Cmd.Jog.ShuttleID].Position.X);
	gMain.Par.Jog.Position.Y := (gVisShuttle.ShuttleInfo[gMain.Cmd.Jog.ShuttleID].Position.Y);
	// Set the jog velocity and Acceleration

	gMain.Cmd.Jog.ShuttleID :=	UINT_TO_USINT(gMain.Par.SelectedIndex); // Selected shuttle
	gMain.Par.Jog.EndVelocity :=  0.0;
	// Pitch and Yaw limit
	MTLookUpTable_0.InX := gVisShuttle.ShuttleInfo[gMain.Cmd.Jog.ShuttleID].Position.Z;
	YawLimit := MTLookUpTable_0.Out;

	// Movement complete
	IF MC_BR_MoveInPlane_Acp6D_0.Done OR MC_BR_MoveShortAxis_Acp6D_0.Done THEN

		MC_BR_MoveShortAxis_Acp6D_0.Execute := FALSE;
		MC_BR_MoveInPlane_Acp6D_0.Execute 	   := FALSE;
	ELSIF EDGENEG(gMain.Cmd.Jog.Left OR gMain.Cmd.Jog.Right OR gMain.Cmd.Jog.Neg OR gMain.Cmd.Jog.Pos)THEN

		MC_BR_ShStop_Acp6D_0.Shuttle := ADR(gShuttleReference[gMain.Cmd.Jog.ShuttleID].Reference);
		MC_BR_ShStop_Acp6D_0.Execute := TRUE;

		// Move left the jog distance
	ELSIF gMain.Cmd.Jog.Left AND((gVisShuttle.ShuttleInfo[gMain.Cmd.Jog.ShuttleID].Position.X - gMain.Cmd.Jog.Distance) > 0.01)THEN

		MC_BR_MoveInPlane_Acp6D_0.Shuttle 	   := ADR(gShuttleReference[gMain.Cmd.Jog.ShuttleID].Reference);
		MC_BR_MoveInPlane_Acp6D_0.Execute 	   := TRUE;
		gMain.Par.Jog.Position.X := 0.045;//(gVisShuttle.ShuttleInfo[gMain.Cmd.Jog.ShuttleID].Position.X - gMain.Cmd.Jog.Distance);
			gMain.Par.Jog.Position.Y :=  gVisShuttle.ShuttleInfo[gMain.Cmd.Jog.ShuttleID].Position.Y;
		MC_BR_MoveInPlane_Acp6D_0.Parameters   :=  gMain.Par.Jog;
		MC_BR_MoveInPlane_Acp6D_0.CommandLabel := 90;

		// Move right the jog distance
	ELSIF gMain.Cmd.Jog.Right AND((gVisShuttle.ShuttleInfo[gMain.Cmd.Jog.ShuttleID].Position.X + gMain.Cmd.Jog.Distance) < 0.239) THEN

		MC_BR_MoveInPlane_Acp6D_0.Shuttle 	   := ADR(gShuttleReference[gMain.Cmd.Jog.ShuttleID].Reference);
		MC_BR_MoveInPlane_Acp6D_0.Execute 	   := TRUE;
		gMain.Par.Jog.Position.X := gAssemblyX_max + 0.015;//0.195;//(gVisShuttle.ShuttleInfo[gMain.Cmd.Jog.ShuttleID].Position.X + gMain.Cmd.Jog.Distance);
		gMain.Par.Jog.Position.Y :=  gVisShuttle.ShuttleInfo[gMain.Cmd.Jog.ShuttleID].Position.Y;
		MC_BR_MoveInPlane_Acp6D_0.Parameters   :=  gMain.Par.Jog;
		MC_BR_MoveInPlane_Acp6D_0.CommandLabel := 91;

		// Move down the jog distance
	ELSIF gMain.Cmd.Jog.Neg AND((gVisShuttle.ShuttleInfo[gMain.Cmd.Jog.ShuttleID].Position.Y - gMain.Cmd.Jog.Distance) > 0.01)THEN

		MC_BR_MoveInPlane_Acp6D_0.Shuttle 	   := ADR(gShuttleReference[gMain.Cmd.Jog.ShuttleID].Reference);
		MC_BR_MoveInPlane_Acp6D_0.Execute 	   := TRUE;
	gMain.Par.Jog.Position.X :=  gVisShuttle.ShuttleInfo[gMain.Cmd.Jog.ShuttleID].Position.X;
		gMain.Par.Jog.Position.Y := 0.045;//(gVisShuttle.ShuttleInfo[gMain.Cmd.Jog.ShuttleID].Position.Y - gMain.Cmd.Jog.Distance);
		MC_BR_MoveInPlane_Acp6D_0.Parameters   :=  gMain.Par.Jog;
		MC_BR_MoveInPlane_Acp6D_0.CommandLabel := 92;

		// Move up the jog distance
	ELSIF gMain.Cmd.Jog.Pos AND((gVisShuttle.ShuttleInfo[gMain.Cmd.Jog.ShuttleID].Position.Y + gMain.Cmd.Jog.Distance) < 0.479)THEN

		MC_BR_MoveInPlane_Acp6D_0.Shuttle 	   := ADR(gShuttleReference[gMain.Cmd.Jog.ShuttleID].Reference);
		MC_BR_MoveInPlane_Acp6D_0.Execute 	   := TRUE;
		gMain.Par.Jog.Position.X :=  gVisShuttle.ShuttleInfo[gMain.Cmd.Jog.ShuttleID].Position.X;
		gMain.Par.Jog.Position.Y := gAssemblyY_max + 0.015;//0.435;//(gVisShuttle.ShuttleInfo[gMain.Cmd.Jog.ShuttleID].Position.Y + gMain.Cmd.Jog.Distance);
		MC_BR_MoveInPlane_Acp6D_0.Parameters   :=  gMain.Par.Jog;
		MC_BR_MoveInPlane_Acp6D_0.CommandLabel := 93;

	ELSIF gMain.Cmd.Jog.RzP AND((gVisShuttle.ShuttleInfo[gMain.Cmd.Jog.ShuttleID].Position.Rz + (gMain.Cmd.Jog.Degrees * 0.017453293)) < 0.136)THEN

		gMain.Par.JogShort.Position.Rx := gVisShuttle.ShuttleInfo[gMain.Cmd.Jog.ShuttleID].Position.Rx;
		gMain.Par.JogShort.Position.Ry := gVisShuttle.ShuttleInfo[gMain.Cmd.Jog.ShuttleID].Position.Ry;
		gMain.Par.JogShort.Position.Z := gVisShuttle.ShuttleInfo[gMain.Cmd.Jog.ShuttleID].Position.Z;
		gMain.Par.JogShort.Position.Rz := (gVisShuttle.ShuttleInfo[gMain.Cmd.Jog.ShuttleID].Position.Rz + (gMain.Cmd.Jog.Degrees * 0.017453293 ));

		MC_BR_MoveShortAxis_Acp6D_0.Shuttle 	 := ADR(gShuttleReference[gMain.Cmd.Jog.ShuttleID].Reference);
		MC_BR_MoveShortAxis_Acp6D_0.Execute 	 := TRUE;
		MC_BR_MoveShortAxis_Acp6D_0.Parameters   :=  gMain.Par.JogShort;
		MC_BR_MoveShortAxis_Acp6D_0.CommandLabel := 94;

	ELSIF gMain.Cmd.Jog.RzN AND(((gVisShuttle.ShuttleInfo[gMain.Cmd.Jog.ShuttleID].Position.Rz - ((gMain.Cmd.Jog.Degrees * 0.017453293))) > -0.136))THEN

		gMain.Par.JogShort.Position.Rx := gVisShuttle.ShuttleInfo[gMain.Cmd.Jog.ShuttleID].Position.Rx;
		gMain.Par.JogShort.Position.Ry := gVisShuttle.ShuttleInfo[gMain.Cmd.Jog.ShuttleID].Position.Ry;
		gMain.Par.JogShort.Position.Z := gVisShuttle.ShuttleInfo[gMain.Cmd.Jog.ShuttleID].Position.Z;
		gMain.Par.JogShort.Position.Rz := (gVisShuttle.ShuttleInfo[gMain.Cmd.Jog.ShuttleID].Position.Rz - (gMain.Cmd.Jog.Degrees * 0.017453293 )); // Convert deg to mRad

		MC_BR_MoveShortAxis_Acp6D_0.Shuttle 	 := ADR(gShuttleReference[gMain.Cmd.Jog.ShuttleID].Reference);
		MC_BR_MoveShortAxis_Acp6D_0.Execute 	 := TRUE;
		MC_BR_MoveShortAxis_Acp6D_0.Parameters   :=  gMain.Par.JogShort;
		MC_BR_MoveShortAxis_Acp6D_0.CommandLabel := 95;

	ELSIF gMain.Cmd.Jog.RxP AND((gVisShuttle.ShuttleInfo[gMain.Cmd.Jog.ShuttleID].Position.Rx + (0.1 * 0.017453293)) < YawLimit)THEN

		gMain.Par.JogShort.Position.Rx := gVisShuttle.ShuttleInfo[gMain.Cmd.Jog.ShuttleID].Position.Rx + (0.1 * 0.017453293);
		gMain.Par.JogShort.Position.Ry := gVisShuttle.ShuttleInfo[gMain.Cmd.Jog.ShuttleID].Position.Ry;
		gMain.Par.JogShort.Position.Z  := gVisShuttle.ShuttleInfo[gMain.Cmd.Jog.ShuttleID].Position.Z;
		gMain.Par.JogShort.Position.Rz := gVisShuttle.ShuttleInfo[gMain.Cmd.Jog.ShuttleID].Position.Rz;

		MC_BR_MoveShortAxis_Acp6D_0.Shuttle 	 := ADR(gShuttleReference[gMain.Cmd.Jog.ShuttleID].Reference);
		MC_BR_MoveShortAxis_Acp6D_0.Execute 	 := TRUE;
		MC_BR_MoveShortAxis_Acp6D_0.Parameters   := gMain.Par.JogShort;
		MC_BR_MoveShortAxis_Acp6D_0.CommandLabel := 96;

	ELSIF gMain.Cmd.Jog.RxN AND((gVisShuttle.ShuttleInfo[gMain.Cmd.Jog.ShuttleID].Position.Rx -((0.1 * 0.017453293)) > -YawLimit))THEN

		gMain.Par.JogShort.Position.Rx := gVisShuttle.ShuttleInfo[gMain.Cmd.Jog.ShuttleID].Position.Rx  - (0.1 * 0.017453293);
		gMain.Par.JogShort.Position.Ry := gVisShuttle.ShuttleInfo[gMain.Cmd.Jog.ShuttleID].Position.Ry;
		gMain.Par.JogShort.Position.Z  := gVisShuttle.ShuttleInfo[gMain.Cmd.Jog.ShuttleID].Position.Z;
		gMain.Par.JogShort.Position.Rz := gVisShuttle.ShuttleInfo[gMain.Cmd.Jog.ShuttleID].Position.Rz; // Convert deg to mRad

		MC_BR_MoveShortAxis_Acp6D_0.Shuttle 	 := ADR(gShuttleReference[gMain.Cmd.Jog.ShuttleID].Reference);
		MC_BR_MoveShortAxis_Acp6D_0.Execute 	 := TRUE;
		MC_BR_MoveShortAxis_Acp6D_0.Parameters   := gMain.Par.JogShort;
		MC_BR_MoveShortAxis_Acp6D_0.CommandLabel := 97;

	ELSIF gMain.Cmd.Jog.RyP AND((gVisShuttle.ShuttleInfo[gMain.Cmd.Jog.ShuttleID].Position.Ry + (0.1 * 0.017453293)) < YawLimit)THEN

		gMain.Par.JogShort.Position.Rx := gVisShuttle.ShuttleInfo[gMain.Cmd.Jog.ShuttleID].Position.Rx;
		gMain.Par.JogShort.Position.Ry := gVisShuttle.ShuttleInfo[gMain.Cmd.Jog.ShuttleID].Position.Ry + (0.1 * 0.017453293);
		gMain.Par.JogShort.Position.Z  := gVisShuttle.ShuttleInfo[gMain.Cmd.Jog.ShuttleID].Position.Z;
		gMain.Par.JogShort.Position.Rz := gVisShuttle.ShuttleInfo[gMain.Cmd.Jog.ShuttleID].Position.Rz;

		MC_BR_MoveShortAxis_Acp6D_0.Shuttle 	 := ADR(gShuttleReference[gMain.Cmd.Jog.ShuttleID].Reference);
		MC_BR_MoveShortAxis_Acp6D_0.Execute 	 := TRUE;
		MC_BR_MoveShortAxis_Acp6D_0.Parameters   := gMain.Par.JogShort;
		MC_BR_MoveShortAxis_Acp6D_0.CommandLabel := 98;

	ELSIF gMain.Cmd.Jog.RyN AND((gVisShuttle.ShuttleInfo[gMain.Cmd.Jog.ShuttleID].Position.Ry -((0.1 * 0.017453293)) > -YawLimit))THEN

		gMain.Par.JogShort.Position.Rx := gVisShuttle.ShuttleInfo[gMain.Cmd.Jog.ShuttleID].Position.Rx;
		gMain.Par.JogShort.Position.Ry := gVisShuttle.ShuttleInfo[gMain.Cmd.Jog.ShuttleID].Position.Ry - (0.1 * 0.017453293);
		gMain.Par.JogShort.Position.Z  := gVisShuttle.ShuttleInfo[gMain.Cmd.Jog.ShuttleID].Position.Z;
		gMain.Par.JogShort.Position.Rz := gVisShuttle.ShuttleInfo[gMain.Cmd.Jog.ShuttleID].Position.Rz; // Convert deg to mRad

		MC_BR_MoveShortAxis_Acp6D_0.Shuttle 	 := ADR(gShuttleReference[gMain.Cmd.Jog.ShuttleID].Reference);
		MC_BR_MoveShortAxis_Acp6D_0.Execute 	 := TRUE;
		MC_BR_MoveShortAxis_Acp6D_0.Parameters   := gMain.Par.JogShort;
		MC_BR_MoveShortAxis_Acp6D_0.CommandLabel := 99;

	ELSIF gMain.Cmd.Jog.Up AND((gVisShuttle.ShuttleInfo[gMain.Cmd.Jog.ShuttleID].Position.Ry + 0.0001) < 0.0041)THEN

		gMain.Par.JogShort.Position.Rx := gVisShuttle.ShuttleInfo[gMain.Cmd.Jog.ShuttleID].Position.Rx;
		gMain.Par.JogShort.Position.Ry := gVisShuttle.ShuttleInfo[gMain.Cmd.Jog.ShuttleID].Position.Ry;
		gMain.Par.JogShort.Position.Z  := gVisShuttle.ShuttleInfo[gMain.Cmd.Jog.ShuttleID].Position.Z + 0.0001;
		gMain.Par.JogShort.Position.Rz := gVisShuttle.ShuttleInfo[gMain.Cmd.Jog.ShuttleID].Position.Rz;

		MC_BR_MoveShortAxis_Acp6D_0.Shuttle 	 := ADR(gShuttleReference[gMain.Cmd.Jog.ShuttleID].Reference);
		MC_BR_MoveShortAxis_Acp6D_0.Execute 	 := TRUE;
		MC_BR_MoveShortAxis_Acp6D_0.Parameters   := gMain.Par.JogShort;
		MC_BR_MoveShortAxis_Acp6D_0.CommandLabel := 100;

	ELSIF gMain.Cmd.Jog.Down AND((gVisShuttle.ShuttleInfo[gMain.Cmd.Jog.ShuttleID].Position.Z - 0.0001) > 0.0009)THEN

		gMain.Par.JogShort.Position.Rx := gVisShuttle.ShuttleInfo[gMain.Cmd.Jog.ShuttleID].Position.Rx;
		gMain.Par.JogShort.Position.Ry := gVisShuttle.ShuttleInfo[gMain.Cmd.Jog.ShuttleID].Position.Ry;
		gMain.Par.JogShort.Position.Z  := gVisShuttle.ShuttleInfo[gMain.Cmd.Jog.ShuttleID].Position.Z - 0.0001;
		gMain.Par.JogShort.Position.Rz := gVisShuttle.ShuttleInfo[gMain.Cmd.Jog.ShuttleID].Position.Rz; // Convert deg to mRad

		MC_BR_MoveShortAxis_Acp6D_0.Shuttle 	 := ADR(gShuttleReference[gMain.Cmd.Jog.ShuttleID].Reference);
		MC_BR_MoveShortAxis_Acp6D_0.Execute 	 := TRUE;
		MC_BR_MoveShortAxis_Acp6D_0.Parameters   := gMain.Par.JogShort;
		MC_BR_MoveShortAxis_Acp6D_0.CommandLabel := 101;

	// Zero the short axes
	ELSIF gMain.Cmd.Jog.Zero THEN

		gMain.Par.JogShort.Position.Rx := 0;
		gMain.Par.JogShort.Position.Ry := 0;
		gMain.Par.JogShort.Position.Z  := 0.001;
		gMain.Par.JogShort.Position.Rz := 0; // Convert deg to mRad

		MC_BR_MoveShortAxis_Acp6D_0.Shuttle 	 := ADR(gShuttleReference[gMain.Cmd.Jog.ShuttleID].Reference);
		MC_BR_MoveShortAxis_Acp6D_0.Execute 	 := TRUE;
		MC_BR_MoveShortAxis_Acp6D_0.Parameters   := gMain.Par.JogShort;
		MC_BR_MoveShortAxis_Acp6D_0.CommandLabel := 102;

		// Clear the command if there is an obstacle
	ELSIF(gVisShuttle.ShuttleInfoVis[gMain.Cmd.Jog.ShuttleID].State = mcACP6D_SH_STATE_OBSTACLE)THEN

		MC_BR_MoveInPlane_Acp6D_0.Execute 	   := FALSE;
		MC_BR_MoveShortAxis_Acp6D_0.Execute := FALSE;
		MC_BR_ShStop_Acp6D_0.Shuttle := ADR(gShuttleReference[gMain.Cmd.Jog.ShuttleID].Reference);
		MC_BR_ShStop_Acp6D_0.Execute := TRUE;

		// Reset the comand if there is an error
	ELSIF MC_BR_MoveInPlane_Acp6D_0.Error OR MC_BR_MoveShortAxis_Acp6D_0.Error THEN

		MC_BR_MoveInPlane_Acp6D_0.Execute 	   := FALSE;
		MC_BR_MoveShortAxis_Acp6D_0.Execute := FALSE;

	END_IF

	IF MC_BR_ShStop_Acp6D_0.Done THEN
			MC_BR_ShStop_Acp6D_0.Execute := FALSE;
	END_IF

END_ACTION
```

#### WeighAct.st
```iecst
ACTION WeighAct:

	CASE stateWeigh OF

		0:
			IF gMain.Status.ShuttlesPresent > 0 THEN
				MC_BR_MoveInPlaneAsync_Acp6D_0.Parameters.AsyncPar[0].Shuttle := ADR(gShuttleReference[0].Reference);
				MC_BR_MoveInPlaneAsync_Acp6D_0.Parameters.AsyncPar[0].X := 0.06;
				MC_BR_MoveInPlaneAsync_Acp6D_0.Parameters.AsyncPar[0].Y := 0.06;
			END_IF

			IF gMain.Status.ShuttlesPresent > 1 THEN
				MC_BR_MoveInPlaneAsync_Acp6D_0.Parameters.AsyncPar[1].Shuttle := ADR(gShuttleReference[1].Reference);
				MC_BR_MoveInPlaneAsync_Acp6D_0.Parameters.AsyncPar[1].X := gAssemblyX_max;
				MC_BR_MoveInPlaneAsync_Acp6D_0.Parameters.AsyncPar[1].Y := gAssemblyY_max;
			END_IF

			IF gMain.Status.ShuttlesPresent > 2 THEN
				MC_BR_MoveInPlaneAsync_Acp6D_0.Parameters.AsyncPar[2].Shuttle := ADR(gShuttleReference[2].Reference);
				MC_BR_MoveInPlaneAsync_Acp6D_0.Parameters.AsyncPar[2].X := gAssemblyX_max;
				MC_BR_MoveInPlaneAsync_Acp6D_0.Parameters.AsyncPar[2].Y := 0.060;
			END_IF

			IF gMain.Status.ShuttlesPresent > 3 THEN
				MC_BR_MoveInPlaneAsync_Acp6D_0.Parameters.AsyncPar[3].Shuttle := ADR(gShuttleReference[3].Reference);
				MC_BR_MoveInPlaneAsync_Acp6D_0.Parameters.AsyncPar[3].X := 0.060;
				MC_BR_MoveInPlaneAsync_Acp6D_0.Parameters.AsyncPar[3].Y := gAssemblyY_max;
			END_IF

			MC_BR_MoveInPlaneAsync_Acp6D_0.Execute 	   := TRUE;
			MC_BR_MoveInPlaneAsync_Acp6D_0.Parameters.Acceleration := gMain.Par.Accel;
			MC_BR_MoveInPlaneAsync_Acp6D_0.Parameters.Velocity := gMain.Par.Velocity;

			IF MC_BR_MoveInPlaneAsync_Acp6D_0.Done THEN
				MC_BR_MoveInPlaneAsync_Acp6D_0.Execute 	   := FALSE;
				stateWeigh := 10;
			END_IF

		10:
			MC_BR_MoveShortAxis_Acp6D_0.Parameters.Position.Rx := 0;
			MC_BR_MoveShortAxis_Acp6D_0.Parameters.Position.Ry := 0;
			MC_BR_MoveShortAxis_Acp6D_0.Parameters.Position.Z  := 0.001;
			MC_BR_MoveShortAxis_Acp6D_0.Parameters.Position.Rz := 0; // Convert deg to mRad

			MC_BR_MoveShortAxis_Acp6D_0.Shuttle 	 := ADR(gShuttleReference[gMain.Par.SelectedIndex].Reference);
			MC_BR_MoveShortAxis_Acp6D_0.Execute 	 := TRUE;
			MC_BR_MoveShortAxis_Acp6D_0.CommandLabel := 102;

			IF MC_BR_MoveShortAxis_Acp6D_0.Done THEN
				MC_BR_MoveShortAxis_Acp6D_0.Execute 	 := FALSE;
				stateWeigh := 20;
			END_IF

		20:
			// Timer for settling time
			TON_0.IN := TRUE;
			TON_0.PT := t#1s;
			IF TON_0.Q THEN
				TON_0.IN := FALSE;
				stateWeigh := 25;
				j := 0;
			END_IF

		25:
			IF j <=(gMain.Status.ShuttlesPresent - 1) THEN
				MC_BR_ShGetPayload_Acp6D_0.Shuttle := ADR(gShuttleReference[j].Reference);
				MC_BR_ShGetPayload_Acp6D_0.Execute := TRUE;

				IF MC_BR_ShGetPayload_Acp6D_0.Done THEN
					TareWeight[j] := (MC_BR_ShGetPayload_Acp6D_0.Payload * 1000);
					j := j+1;
					MC_BR_ShGetPayload_Acp6D_0.Execute := FALSE;
					IF j = (gMain.Status.ShuttlesPresent) THEN
						stateWeigh := 30;
						j := 0;
					END_IF
				END_IF
			END_IF

		30:

			IF j <=(gMain.Status.ShuttlesPresent - 1) THEN
				MC_BR_ShGetPayload_Acp6D_0.Shuttle := ADR(gShuttleReference[j].Reference);
				MC_BR_ShGetPayload_Acp6D_0.Execute := TRUE;

				IF MC_BR_ShGetPayload_Acp6D_0.Done THEN
					IF m < 500 THEN
						AverageWeightShtl[j,m] := (MC_BR_ShGetPayload_Acp6D_0.Payload * 1000)- TareWeight[j];;
						m := m +1;
					ELSE
						m := 0;
					END_IF

					j := j+1;
					MC_BR_ShGetPayload_Acp6D_0.Execute := FALSE;
					IF j = (gMain.Status.ShuttlesPresent) THEN
						stateWeigh := 40;
						j := 0;
					END_IF
				END_IF
			END_IF

			// calculate average for each shuttle
			FOR l := 0 TO 3 DO
				// Make sure the sum is zeroed
				AverageWeightShtSum[l] := 0;
				// Sum all the values for each shuttle
				FOR k := 0 TO 499 DO
					AverageWeightShtSum[l] :=	AverageWeightShtSum[l] + AverageWeightShtl[l,k];
				END_FOR
			END_FOR
			// Calculate the average
			gMain.Status.Weight[j] :=	AverageWeightShtSum[j]/500;

		40:

			IF (visSelectedTab <> 2)THEN
				MainStep                                :=    MAIN_READY;
				stateWeigh := 0;
			ELSIF(gMain.Cmd.Tare)THEN
				stateWeigh := 25;
			ELSE
				stateWeigh := 30;
			END_IF

	END_CASE

END_ACTION
```

#### RecoverAct.st
```iecst
ACTION RecoverAct:

	MC_BR_ShRecover_Acp6D_0.Shuttle := ADR(gShuttleReference[gMain.Cmd.Jog.ShuttleID].Reference);
	MC_BR_ShRecover_Acp6D_0.Execute := TRUE;

	IF MC_BR_ShRecover_Acp6D_0.Done THEN
		MC_BR_ShRecover_Acp6D_0.Execute := FALSE;
		MainStep          := MAIN_READY;
	ELSIF MC_BR_ShRecover_Acp6D_0.Error THEN
		MC_BR_ShRecover_Acp6D_0.Execute := FALSE;
		MainStep          := MAIN_ERROR;
	END_IF

	stateRecover

END_ACTION
```

### Program Logical/Macro (IEC)

#### Main.st - Init, cyclic, exit code
```iecst
PROGRAM _INIT
	(* Insert code here *)

	MacroName := 'Demo';
	inc			:= 0;
	MC_BR_MacroCreate_Acp6D_0.Assembly := ADR(gAssembly6D_1);
	MC_BR_AsmPowerOn_Acp6D_0.Assembly	:= ADR(gAssembly6D_1);
	MC_BR_AsmReadStatus_0.Assembly		:= ADR(gAssembly6D_1);
	MC_BR_MacroDelete_0.Assembly		:= ADR(gAssembly6D_1);
	MC_BR_AsmGetShuttle_0.Assembly		:= ADR(gAssembly6D_1);
	MC_BR_MoveInPlaneAsync_Acp6D_0.Assembly := ADR(gAssembly6D_1);

END_PROGRAM

PROGRAM _CYCLIC

	Cmd.Start := gCreateDemo;

	IF MacroState < C_NEXT_COMMAND_05 THEN
		visMacroStatus := 'Waiting';
		visLockRun := FALSE;
	ELSIF MacroState >= C_NEXT_COMMAND_05 AND MacroState < C_REMAKE_DEMO_MACRO_70 THEN
		visMacroStatus := 'Creating Demo Marco';
		visLockRun := FALSE;
	ELSIF MacroState = C_REMAKE_DEMO_MACRO_70 THEN
		visMacroStatus := 'Ready';
		visLockRun := TRUE;
	ELSIF MacroState > C_RUN_DEMO_MACRO_80 OR MacroState <= C_RE_RUN_85 THEN
		visMacroStatus := 'Runing Macro';
		visLockRun := FALSE;
	END_IF

	CASE MacroState OF

		C_WAIT_00:

			ResetMacroFubs;

			IF(Cmd.Start)THEN
				Cmd.Start := FALSE;
				command := 0;
				MacroState := C_READ_STATUS_01;
				MC_BR_AsmReadStatus_0.Enable := TRUE;
			END_IF;

		C_READ_STATUS_01:

			IF(MC_BR_AsmReadStatus_0.Valid)THEN
				IF 	gCreateDemo THEN
					MacroName := 'Demo';
					gCreateDemo := FALSE;
					DemoAct;
				END_IF
				IF(MC_BR_AsmReadStatus_0.AssemblyDisabled)THEN
					MacroState := C_POWER_ON_02;
				ELSIF(MC_BR_AsmReadStatus_0.AssemblyReady)THEN
					MacroState := C_CREATE_03;
				END_IF;
			END_IF;

		C_POWER_ON_02:

			MC_BR_AsmPowerOn_Acp6D_0.Execute := TRUE;

			IF(MC_BR_AsmPowerOn_Acp6D_0.Done)THEN
				MC_BR_AsmPowerOn_Acp6D_0.Execute := FALSE;
				MacroState := C_CREATE_03;
			END_IF;

		C_CREATE_03:

			MC_BR_MacroCreate_Acp6D_0.Parameters.Name := MacroName;
			int_to_str := USINT_TO_STRING(inc);
			brsstrcat(ADR(MC_BR_MacroCreate_Acp6D_0.Parameters.Name),ADR(int_to_str));
			TempName := MC_BR_MacroCreate_Acp6D_0.Parameters.Name;
			MC_BR_MacroCreate_Acp6D_0.Execute := TRUE;

			IF(MC_BR_MacroCreate_Acp6D_0.Done)THEN
				MC_BR_MacroCreate_Acp6D_0.Execute := FALSE;
				MacroState := C_NEXT_COMMAND_05;
				MacroSh[inc] := MC_BR_MacroCreate_Acp6D_0.MacroShuttle;
			ELSIF MC_BR_MacroCreate_Acp6D_0.ErrorID = -1065811716 THEN
					MC_BR_MacroCreate_Acp6D_0.Execute := FALSE;
					MacroState := C_DELETE_04;
			END_IF;

		C_DELETE_04:

			MC_BR_MacroDelete_0.Name := MacroName;
			MC_BR_MacroDelete_0.Command :=	mcACP6D_MACRO_DELETE_SPECIFIC;
			MC_BR_MacroDelete_0.Execute := TRUE;

			IF(MC_BR_MacroDelete_0.Done)THEN
				MC_BR_MacroDelete_0.Execute := FALSE;
				Cmd.Start := FALSE;
				MacroState := C_WAIT_00;
			ELSIF  MC_BR_MacroDelete_0.ErrorID = -1065811714  THEN
				MC_BR_MacroDelete_0.Execute := FALSE;
				Cmd.Start := FALSE;
				MacroState := C_WAIT_00;
			END_IF

		C_NEXT_COMMAND_05:

			IF gMacro[command].CommandType = 60 THEN
				MacroState := gMacro[command].CommandType;
			ELSE
				MacroState := gMacro[command].CommandType;
			END_IF

		C_MOVE_IN_PLANE_010:

			MC_BR_MoveInPlane_Acp6D_0.Shuttle 	 := ADR(MacroSh[inc]);;
			MC_BR_MoveInPlane_Acp6D_0.Parameters := gMacro[command].MovePlane;
			MC_BR_MoveInPlane_Acp6D_0.Execute 	 := TRUE;

			IF(MC_BR_MoveInPlane_Acp6D_0.Acknowledge)THEN
				MC_BR_MoveInPlane_Acp6D_0.Execute := FALSE;
				command := command + 1;
				MacroState := C_NEXT_COMMAND_05;
			END_IF;

		C_MOVE_IN_PLANE_ASYNC_015:

			MC_BR_MoveInPlaneAsync_Acp6D_0.Parameters	:= gMacro[command].MoveAsync;
			MC_BR_MoveInPlaneAsync_Acp6D_0.Execute 	:= TRUE;

			IF(MC_BR_MoveInPlaneAsync_Acp6D_0.Acknowledge)THEN
				MC_BR_MoveInPlaneAsync_Acp6D_0.Execute := FALSE;
				command := command + 1;
				MacroState := C_NEXT_COMMAND_05;
			END_IF;

		C_MOVE_IN_6D_PLANE_020:

			MC_BR_Move6D_Acp6D_0.Shuttle 	:= ADR(MacroSh[inc]);
			MC_BR_Move6D_Acp6D_0.Parameters	:= gMacro[command].Move6D;
			MC_BR_Move6D_Acp6D_0.Execute 	:= TRUE;

			IF(MC_BR_Move6D_Acp6D_0.Acknowledge)THEN
				MC_BR_Move6D_Acp6D_0.Execute := FALSE;
				command := command + 1;
				MacroState := C_NEXT_COMMAND_05;
			END_IF;

		C_MOVE_ARC_025:

			MC_BR_MoveArc_Acp6D_0.Shuttle 		:= ADR(MacroSh[inc]);
			MC_BR_MoveArc_Acp6D_0.Parameters	:= gMacro[command].MoveArc;
			MC_BR_MoveArc_Acp6D_0.Execute 		:= TRUE;

			IF(MC_BR_MoveArc_Acp6D_0.Acknowledge)THEN
				MC_BR_MoveArc_Acp6D_0.Execute := FALSE;
				command := command + 1;
				MacroState := C_NEXT_COMMAND_05;
			END_IF;

		C_SAVE_60:

			MC_BR_MacroSave_0.Shuttle := ADR(MacroSh[inc]);
			MC_BR_MacroSave_0.Execute := TRUE;

			IF(MC_BR_MacroSave_0.Done)THEN
				ExistingMacroNames[inc] := TempName;
				MC_BR_MacroSave_0.Execute := FALSE;
				MacroState := C_REMAKE_DEMO_MACRO_70;
				command := 0;
				inc := inc+1;
				i := 0;
			ELSIF(MC_BR_MacroSave_0.Error AND Clear)THEN
				MC_BR_MacroSave_0.Execute := FALSE;
				MacroState := C_RESET_100;
			END_IF;

		C_REMAKE_DEMO_MACRO_70:

			// Recreate the demo macro for all shuttles (MAX 4 in this action)
			IF(inc < gMain.Status.ShuttlesPresent)THEN
				MacroState := C_READ_STATUS_01;
			END_IF

			IF RunMacro THEN
				RunMacro := FALSE;
				MacroState := C_RUN_DEMO_MACRO_80;
			END_IF

		C_RUN_DEMO_MACRO_80:

			MC_BR_MacroRun_0.Shuttle := ADR(gShuttleReference[0].Reference);
			MC_BR_MacroRun_0.Execute := TRUE;
			MC_BR_MacroRun_0.Name	:= ExistingMacroNames[0];

			IF(MC_BR_MacroRun_0.Acknowledge)THEN
				MC_BR_MacroRun_0.Execute := FALSE;
				MacroState := C_RUN_DEMO_MACRO_81;
			END_IF;

		C_RUN_DEMO_MACRO_81:

			IF gMain.Status.ShuttlesPresent > 3 THEN
				MC_BR_MacroRun_0.Shuttle := ADR(gShuttleReference[3].Reference);
				MC_BR_MacroRun_0.Execute := TRUE;
				MC_BR_MacroRun_0.Name	:= ExistingMacroNames[3];

				IF(MC_BR_MacroRun_0.Acknowledge)THEN
					MC_BR_MacroRun_0.Execute := FALSE;
					MacroState := C_RUN_DEMO_MACRO_82;
				END_IF;
			ELSE
				MacroState := C_RUN_DEMO_MACRO_82;
			END_IF

		C_RUN_DEMO_MACRO_82:

			IF gMain.Status.ShuttlesPresent > 2 THEN
				MC_BR_MacroRun_0.Shuttle := ADR(gShuttleReference[2].Reference);
				MC_BR_MacroRun_0.Execute := TRUE;
				MC_BR_MacroRun_0.Name	:= ExistingMacroNames[2];

				IF(MC_BR_MacroRun_0.Acknowledge)THEN
					MC_BR_MacroRun_0.Execute := FALSE;
					MacroState := C_RUN_DEMO_MACRO_83;
				END_IF;
			ELSE
				MacroState := C_RUN_DEMO_MACRO_83;
			END_IF

		C_RUN_DEMO_MACRO_83:

			IF gMain.Status.ShuttlesPresent > 1 THEN
				MC_BR_MacroRun_0.Shuttle := ADR(gShuttleReference[1].Reference);
				MC_BR_MacroRun_0.Execute := TRUE;
				MC_BR_MacroRun_0.Name	:= ExistingMacroNames[1];

				IF(MC_BR_MacroRun_0.Acknowledge)THEN
					MC_BR_MacroRun_0.Execute := FALSE;
					MacroState := C_RE_RUN_85;
				END_IF;
			ELSE
				MacroState := C_RE_RUN_85;
			END_IF

		C_RE_RUN_85:

			IF(gVisShuttle.ShuttleInfoVis[0].State <> mcACP6D_SH_STATE_MOTION)AND(gVisShuttle.ShuttleInfoVis[1].State <> mcACP6D_SH_STATE_MOTION)AND(gVisShuttle.ShuttleInfoVis[2].State <> mcACP6D_SH_STATE_MOTION)AND(gVisShuttle.ShuttleInfoVis[3].State <> mcACP6D_SH_STATE_MOTION)THEN
				MacroState := C_REMAKE_DEMO_MACRO_70;
			END_IF

			IF ReRun THEN
				RunMacro := TRUE;
			END_IF

		C_CLEARMACRO_90:

			MC_BR_MacroClear_0.Shuttle := ADR(MacroSh[inc]);
			MC_BR_MacroClear_0.Execute := TRUE;

			IF(MC_BR_MacroClear_0.Done)THEN
				MC_BR_MacroClear_0.Execute := FALSE;
				MacroState := C_WAIT_00;
			END_IF;

		C_RESET_100:

			IF(Cmd.Reset)THEN
				MacroState := C_WAIT_00;
				Cmd.Start := FALSE;
				Cmd.Reset := FALSE;
				Cmd.Stop := FALSE;
				Clear := FALSE;
			END_IF;

	END_CASE;

	MC_BR_AsmPowerOn_Acp6D_0();
	MC_BR_MacroCreate_Acp6D_0();
	MC_BR_MoveInPlane_Acp6D_0();
	MC_BR_MoveInPlaneAsync_Acp6D_0();
	MC_BR_Move6D_Acp6D_0();
	MC_BR_MoveArc_Acp6D_0();
	MC_BR_AsmReadStatus_0();
	MC_BR_MacroSave_0();
	MC_BR_MacroClear_0();
	MC_BR_MacroDelete_0();
	MC_BR_MacroRun_0();
	MC_BR_AsmGetShuttle_0();
END_PROGRAM

PROGRAM _EXIT
	(* Insert code here *)

END_PROGRAM
```

#### Types.typ - Local data types
```iecst
TYPE
	Macro_typ : 	STRUCT
		Move6D : McAcp6DMove6DParType;
		MoveAsync : McAcp6DMoveInPlaneAsyncParType;
		MoveArc : McAcp6DArcParType;
		MovePlane : McAcp6DInPlaneParType;
		CommandType : USINT;
		ShuttleID : UINT;
	END_STRUCT;
END_TYPE
```
